10:	IF ip_state = BYTE#3 THEN (* Bei IP_Control anmelden *)
		url_length := LEN(domain_copy);
		char_count := 17 + url_length; (* sendebuffer initialisieren *)
		FOR i := 0 TO char_count DO
			S_BUF.BUFFER[i] := BYTE#00;
		END_FOR;
		tid := UINT_TO_BYTE(BYTE_TO_UINT(tid) + UINT#1);
		S_BUF.BUFFER[01] := tid; (* Transaction ID lowbyte *)
		S_BUF.BUFFER[02] := BYTE#16#01; (* Flags: highbyte *)
		S_BUF.BUFFER[05] := BYTE#16#01; (* Questions: lowbyte *)
		i := url_length + 12;	(* den servernamen von hinten nach vorne bearbeiten *)
		char_count := 0;
		WHILE i > 12 DO
			char := CODE(STR:=domain_copy,POS:=i - 12);
			IF char = BYTE#46 THEN (* prüfe auf haupt/sub domänen namens-teiler "." *)
				S_BUF.BUFFER[i] := INT_TO_BYTE(char_count); (* anstelle des teilers "." wird die länge des erkannten haupt/sub domänennames eingetragen *)
				char_count := 0;
			ELSE
				S_BUF.BUFFER[i] := char; (* char in buffer eintragen *)
				char_count := char_count + 1; (* anzahl char zählen *)
			END_IF;
			i := i - 1;
		END_WHILE;
		S_BUF.BUFFER[i] := INT_TO_BYTE(char_count); (* längenangabe des ganz linken (ersten) domänennamens eintragen *)
		i := url_length + 15; (* position hinter dem servernamen *)
		S_BUF.BUFFER[i] := BYTE#01; (* Type: A Hostaddress lowbyte *)
		i := i + 2;
		S_BUF.BUFFER[i] := BYTE#01; (* Class: IN lowbyte *)
		i := i + 1;
		(* IP Datenverkehr einrichten *)
		IP_C.C_PORT := WORD#53; (* Portnummer eintragen *)
		IP_C.C_IP := IP4_DNS; (* IP eintragen *)
		IP_C.C_MODE := BYTE#1; (* Mode: UDP+AKTIV+PORT+IP *)
		IP_C.C_ENABLE := TRUE; (* Verbindungsaufbau freigeben *)
		IP_C.TIME_RESET := TRUE; (* Zeitueberwachung rücksetzen *)
		IP_C.R_OBSERVE  := TRUE; (* Datenempfang ueberwachen *)
		S_BUF.SIZE := INT_TO_UINT(i); (* sendelänge eintragen *)
		R_BUF.SIZE := UINT#0; (* Empfangslänge rücksetzen *)
		state := 30;

        		(*####################  DEBUG-MESSAGE  ###################################*)
        		(*IF _debug_enable THEN
            		LOG_CL.NEW_MSG := 'DNS: S10 SEND';
            		LOG_MSG();
        		END_IF;*)
        		(*########################################################################*)
	END_IF;

30:	IF IP_C.ERROR <> DWORD#00 THEN
		ERROR := IP_C.ERROR;
		state := 99;
        		(*####################  DEBUG-MESSAGE  ###################################*)
        		(*IF _debug_enable THEN
            		LOG_CL.NEW_MSG := 'DNS: S30 ERROR ~1';
            		LOG_CL.PRINTF[1]  := DWORD_TO_STRING(ERROR);
            		LOG_MSG();
        		END_IF;*)
        		(*########################################################################*)

	ELSIF (S_BUF.SIZE = UINT#0) AND (tid = R_BUF.BUFFER[1]) AND (R_BUF.SIZE >= INT_TO_UINT(34 + url_length)) THEN	(* prüfe ob antwort telegramm die richtige Transaction-ID und mindestlänge hat *)
		ERROR := BYTE_TO_DWORD(R_BUF.BUFFER[3] AND BYTE#2#0000_1111); (* prüfe Return code der Flags. 4 bits *)
		IF ERROR = DWORD#00 THEN
			anc := R_BUF.BUFFER[7]; (* Anzahl der Answer-RR *)
			IP_C.R_OBSERVE := FALSE; (* Datenempfang ueberwachen *)
			state := 40;
		ELSE
			state := 99;
		END_IF;
	END_IF;

40:	IF anc > 0 THEN
		anc := anc - 1;
		WHILE i < R_BUF.SIZE DO
			x := R_BUF.BUFFER[i];
			IF rr_stop = FALSE THEN
				IF x > BYTE#63 THEN (* zeiger auf namen *)
					i := i + 1;
					rr_stop := TRUE;
				ELSIF x= BYTE#0 THEN (* namens ende *)
					rr_stop := TRUE;
				ELSE
					i := i + x; (* namen *)
				END_IF;
				i := i + 1;
			ELSE
				rr_stop := FALSE;
				IF R_BUF.BUFFER[i+1] = BYTE#1 AND R_BUF.BUFFER[i+3] = BYTE#1 THEN (* Type A / Class IN *)
					i := i + 4;
					ttl_tmp := DWORD_OF_BYTE(R_BUF.BUFFER[i],R_BUF.BUFFER[i+1],R_BUF.BUFFER[i+2],R_BUF.BUFFER[i+3]); (* Time to live *)
					i := i + 6;
					IF ttl_tmp >= ttl_last THEN (* TTL ist länger *)
						ttl_last := ttl_tmp;
						IP4 := DWORD_OF_BYTE(R_BUF.BUFFER[i],R_BUF.BUFFER[i+1],R_BUF.BUFFER[i+2],R_BUF.BUFFER[i+3]); (* IP-Adresse *)
					END_IF;
					i := i + 4;
				ELSE
					i := i + 9;
					i := i + R_BUF.BUFFER[i] + 1; (* offset zu nächsten Block *)
				END_IF;
				EXIT;
			END_IF;
		END_WHILE;
	ELSE
		IF IP4 > DWORD#0 THEN (* gültige RR mit IP gefunden *)
			DONE := TRUE;
            		(*####################  DEBUG-MESSAGE  ###################################*)
            		(*IF _debug_enable THEN
                			LOG_CL.NEW_MSG := 'DNS: S40 OK';
                			LOG_MSG();
            		END_IF;*)
            		(*########################################################################*)
		ELSE
			ERROR := DWORD#255; (* Daten fehlerhaft - keine IP-Adresse vorhanden *)
		END_IF;
		state := 99;
	END_IF;

99:	R_BUF.SIZE := UINT#0; (* Empfangslänge rücksetzen *)
	ip_state := BYTE#4; (* Abmelden *)
	state := 00;

END_CASE;

activate_last := ACTIVATE; (* letzten Status sichern zur Flankenerkennung *)
IP_FIFO(FIFO:=IP_C.FIFO,STATE:=ip_state,ID:=ip_id); (* IP_FIFO *)

(* revision history

ks	18. oct. 2008	rev 1.0
	original version

ks	20. oct. 2009	rev 1.1
	unbenutzten code entfernt, all buffer base 0

ks	20. dec. 2010	rev 1.2
	parsing nach rfc1305

ks	26. jul. 2011	rev 1.3
	verbesserte ip-auswertung , neue fehlermeldung
*)


(*----------------------------------------------------------------------------------------------------------------*)
(* Flags: 0x0100 (Standard query)                                                                                            *)
(* 0... .... .... .... = Response: Message is a query                                                                   *)
(* .000 0... ....  = Opcode: Standard query (0)                                                                          *)
(* .... ..0. .... .... = Truncated: Message is not truncated                                                          *)
(* .... ...1 .... .... = Recursion desired: Do query recursively                                                    *)
(* .... .... .0.. .... = Z: reserved (0)                                                                                                  *)
(* .... .... ...0 .... = Non-authenticated data OK: Non-authenticated data is unacceptable *)
(*-----------------------------------------------------------------------------------------------------------------*)

(*      0  1  2  3  4  5  6  7  8  9  0  1  2  3  4  5  *)
(*    +--+--+--+--+--+--+--+--+--+--+--+--+--+--+--+--+ *)
(*    |                      ID                       | idx: 0/1   *)
(*    +--+--+--+--+--+--+--+--+--+--+--+--+--+--+--+--+ *)
(*    |QR|   Opcode  |AA|TC|RD|RA|   Z    |   RCODE   | idx: 2/3   *)
(*    +--+--+--+--+--+--+--+--+--+--+--+--+--+--+--+--+ *)
(*    |                    QDCOUNT                    | idx: 4/5   *)
(*    +--+--+--+--+--+--+--+--+--+--+--+--+--+--+--+--+ *)
(*    |                    ANCOUNT                    | idx: 6/7   *)
(*    +--+--+--+--+--+--+--+--+--+--+--+--+--+--+--+--+ *)
(*    |                    NSCOUNT                    | idx: 8/9   *)
(*    +--+--+--+--+--+--+--+--+--+--+--+--+--+--+--+--+ *)
(*    |                    ARCOUNT                    | idx: 10/11 *)
(*    +--+--+--+--+--+--+--+--+--+--+--+--+--+--+--+--+ *)

(*
Errorcodes  Description	References 
000	No error. 		 	The request completed successfully.
001	Format error. 		The name server was unable to interpret the query. 
002	Server failure.  	The name server was unable to process this query due to a problem with the name server. 
003	Name Error. 	 	Meaningful only for responses from an authoritative name server, this code signifies that the domain name referenced in the query does not exist.
004	Not Implemented. 	The name server does not support the requested kind of query.
005	Refused. 			The name server refuses to perform the specified operation for policy reasons.
  						 For example, a name server may not wish to provide the information to the particular requester, or a name server may not wish to perform a particular operation (e.g., zone transfer) for particular data.
006	YXDomain.			Name Exists when it should not. 
007	YXRRSet. RR			Set Exists when it should not. 
008	NXRRSet. RR			Set that should exist does not. 
009	NotAuth.			Server Not Authoritative for zone. 
010	NotZone,			Name not contained in zone. 
255	Timeout				No Response  
   

beispiel einer DNS Request von google.at
ein request mit 3 Answer-Blocks


Domain Name System (response)
[Request In: 3]
[Time: 0.027533000 seconds]
Transaction ID: 0x5e1a
Flags: 0x8180 (Standard query response, No error)
1... .... .... .... = Response: Message is a response
.000 0... .... .... = Opcode: Standard query (0)
.... .0.. .... .... = Authoritative: Server is not an authority for domain
.... ..0. .... .... = Truncated: Message is not truncated
.... ...1 .... .... = Recursion desired: Do query recursively
.... .... 1... .... = Recursion available: Server can do recursive queries
.... .... .0.. .... = Z: reserved (0)
.... .... ..0. .... = Answer authenticated: Answer/authority portion was not authenticated
.... .... .... 0000 = Reply code: No error (0)
Questions: 1
Answer RRs: 3
Authority RRs: 0
Additional RRs: 0

Queries
google.at: type A, class IN
Name: google.at
Type: A (Host address)
Class: IN (0x0001)

Answers
google.at: type A, class IN, addr 72.14.221.104
Name: google.at
Type: A (Host address)
Class: IN (0x0001)
Time to live: 19 minutes, 9 seconds
Data length: 4
Addr: 72.14.221.104

google.at: type A, class IN, addr 66.249.93.104
Name: google.at
Type: A (Host address)
Class: IN (0x0001)
Time to live: 19 minutes, 9 seconds
Data length: 4
Addr: 66.249.93.104

google.at: type A, class IN, addr 216.239.59.104
Name: google.at
Type: A (Host address)
Class: IN (0x0001)
Time to live: 19 minutes, 9 seconds
Data length: 4
Addr: 216.239.59.104
*)

END_FUNCTION_BLOCK

// ---- oscat_basic/POUs/String/CHR_TO_STRING.TcPOU
FUNCTION CHR_TO_STRING : STRING(1)
VAR_INPUT
	C : BYTE;
END_VAR
VAR
	PT : POINTER TO BYTE;
END_VAR

(*
version 1.3	17. dec. 2008
programmer 	hugo
tested by	oscat

CHR creates a character from a byte input and stuffs it in a one character length string.

*)

PT := ADR(CHR_TO_STRING);
PT^ := C;
pt := pt + 1;
pt^ := 0;

(* revision history
hm	16 jan 2007		rev 1.0
	original version

hm	4. feb. 2008	rev 1.1
	return string would not be terminated properly

hm	29. mar. 2008	rev 1.2
	changed STRING to STRING(1)

hm	17. dec. 2008	rev 1.3
	changed name of function from chr to chr_to_string
*)

END_FUNCTION

// ---- beckhoff_network/POUs/DEMO/FTP_CLIENT_DEMO.TcPOU
PROGRAM FTP_CLIENT_DEMO
VAR
	FTP_CLIENT: FTP_CLIENT;
	ftp_activate: BOOL;
	ftp_done: BOOL;
	ftp_busy: BOOL;
	ftp_error_c: DWORD;
	ftp_error_t: BYTE;
	ftp_url: STRING := 'ftp://581920:123456@oscat.atwebpages.com:2000/subordner/';
	ftp_filename: STRING := '0100kb.bin';
	ftp_download: BOOL := TRUE;
	ftp_activ: BOOL := FALSE;
	file_delete: BOOL := FALSE;
	ftp_timeout: TIME := T#30s;
	zeit : TIME := T#30s;
	stop: BOOL;
	start: BOOL :=TRUE ;
	reset: BOOL;
	error: DWORD;
	ok: DWORD;
	CLK_PRG_1: CLK_PRG;
	COUNT_DR_1: COUNT_DR;
	COUNT_DR_2: COUNT_DR;
END_VAR
VAR // added by the converter: edge detectors and wires of the graphical bodies
    _w1, _w2 : ANY;
END_VAR

ftp_client(
    ACTIVATE := ftp_activate,
    FILENAME := ftp_filename,
    FTP_URL := ftp_url,
    FTP_DOWNLOAD := ftp_download,
    FTP_ACTIV := ftp_activ,
    FILE_DELETE := file_delete,
    TIMEOUT := ftp_timeout,
    DNS_IP4 := _w1,
    PLC_IP4 := _w2);
ftp_done := ftp_client.DONE;
ftp_busy := ftp_client.BUSY;
ftp_error_c := ftp_client.ERROR_C;
ftp_error_t := ftp_client.ERROR_T;
CLK_PRG_1(_in1 := zeit); // CLK_PRG
ftp_activate := CLK_PRG_1._out1 AND NOT stop AND start OR reset;
stop := ftp_error_t <> 0;
COUNT_DR_1(_in3 := stop); // COUNT_DR
error := COUNT_DR_1._out1;
COUNT_DR_2(_in3 := ftp_done); // COUNT_DR
ok := COUNT_DR_2._out1;
_w1 := DWORD_OF_BYTE(8, 8, 8, 8);
_w2 := DWORD_OF_BYTE(10, 145, 72, 57);

END_PROGRAM

// ---- beckhoff_network/POUs/NETWORK/FTP_CLIENT.TcPOU
FUNCTION_BLOCK FTP_CLIENT
VAR_INPUT
	ACTIVATE : BOOL;
	FILENAME : STRING;
	FTP_URL : STRING(STRING_LENGTH);
	FTP_DOWNLOAD : BOOL;
	FTP_ACTIV : BOOL;
	FILE_DELETE : BOOL;
	TIMEOUT : TIME;
	DNS_IP4 : DWORD;
	PLC_IP4 : DWORD;
END_VAR
VAR_OUTPUT
	DONE : BOOL;
	BUSY : BOOL;
	ERROR_C : DWORD;
	ERROR_T : BYTE;
END_VAR
VAR
	IP_C1 : IP_C; (* IP_Control Verwaltungsstruktur *)
	IP_C2 : IP_C; (* IP_Control Verwaltungsstruktur *)
	S_BUF1 : NETWORK_BUFFER;
	S_BUF2 : NETWORK_BUFFER;
	R_BUF1 : NETWORK_BUFFER;
	R_BUF2 : NETWORK_BUFFER;
	URL_DATA : url;
	DNS_CLIENT : DNS_CLIENT;
	IPC1 : IP_CONTROL;
	IPC2 : IP_CONTROL;
	FS : FILE_SERVER;
	FSD : FILE_SERVER_DATA;

	activate_last : BOOL;
	step : INT;
	snd_step : INT;
	snd_text :	STRING(STRING_LENGTH);
	rcv_text :	STRING(STRING_LENGTH);
	rcv_state : INT;
	TON_WAIT : TON;
	last_step : INT;
	next_step : INT;
	idx1 : INT;
	idx2 : INT;
	str1 : STRING(STRING_LENGTH);
	str2 : STRING(STRING_LENGTH);
	ftp_path : STRING;
	byar : ARRAY [0..5] OF BYTE;
	dw_tmp : DWORD;
	w_tmp : WORD;
	fpd : FILE_PATH_DATA;
	timeout2 : TIME;
	timeout3 : TIME;
	ftp_file_size : UDINT;
	ip_c1_red_disable : BOOL; (* IP_CONTROL 1 - Remote Disconnect Error unterdrücken *)
	ip_c2_red_disable : BOOL; (* IP_CONTROL 1 - Remote Disconnect Error unterdrücken *)

	(*LOG_MSG : LOG_MSG;
	_debug_enable : BOOL := FALSE;*)

END_VAR
(*
version 1.2		11.may 2011
programmer		ks
tested by			ks

FTP_CLIENT dient zum senden und empfangen von dateien von einem FTP-Server.



110 Restart marker reply 										Markierung für Wiederaufnahme der Übertragung 
120 Service ready in x minutes 									Dienst steht in x Minuten zu Verfügung 
125 Data connection already open; 								transfer starting Datenverbindung besteht bereits; beginne mit der Übertragung 
150 File status okay; about to open data connection 					Dateistatus OK; Datenverbindung wird aufgebaut 
200 Command okay 											Befehl OK 
202 Command not implemented 									Befehl nicht implementiert 
211   														Antwort für Systemstatus oder Hilfefunktion des Systems 
212   														Verzeichnisstatus 
213   														Dateistatus 
214   														Meldung der Hilfefunktion 
215 NAME system type 										Angabe des Systemtyps 
220 Service ready for new user 									Dienst bereit für neuen Benutzer 
221 Service closing control connection 							Steuerverbindung des Dienstes wird getrennt; Benutzer wird abgemeldet 
225 Data connection open; no transfer in progress 					Datenverbindung hergestellt; derzeit keine Übertragung 
226 Closing data connection. Requested file action successful 		Datenverbindung wird getrennt 
227 Entering Passive Mode 										Passiver Modus aktiviert 
230 User logged in, proceed 									Benutzer angemeldet, bitte fortfahren 
250 Requested file action okay, completed 						Angeforderter Vorgang OK, beendet 
257 "PATH" created 											"PFAD" wurde erstellt 
331 User name okay, need password 							Benutzername OK, Kennwort erforderlich 
332 Need account for login 										Benutzerkonto zur Anmeldung erforderlich 
350 Requested file action pending further information 				Mehr Informationen für Dateivorgang erforderlich 
421 Service not available, closing control connection 				Dienst nicht verfügbar, Steuerverbindung wird getrennt 
425 Can't open data connection 									Datenverbindung kann nicht hergestellt werden 
426 Connection closed; transfer aborted Verbindung getrennt; 		Übertragung abgebrochen 
450 Requested file action not taken; File unavailable 				Angeforderter Dateivorgang wurde nicht ausgeführt; Datei nicht verfügbar 
451 Requested action aborted: local error in processing 				Angeforderter Vorgang abgebrochen: Lokaler Fehler bei der Bearbeitung 
452 Requested action not taken; Insufficient storage space in system 	Angeforderter Vorgang nicht ausgeführt; Nicht genügend Speicherplatz auf System 
500 Syntax error 												Befehl nicht erkannt 
501 Syntax error in parameters or arguments 						Syntaxfehler bei den Parametern 
502 Command not implemented 									Befehl nicht implementiert 
503 Bad sequence of commands 								Ungültige Befehlsabfolge 
504 Command not implemented for that parameter 					Befehl für diesen Parameter nicht implementiert 
530 Not logged in 												Nicht angemeldet 
532 Need account for storing files 								Zum Speichern von Dateien Anmeldung erforderlich 
550 Requested file action not taken; File unavailable Angeforderter 	Dateivorgang wurde nicht ausgeführt; Datei nicht verfügbar 
551 Requested action aborted: page type unknown 					Angeforderter Vorgang abgebrochen: Unbekannter Seitentyp 
552 Requested file action aborted: Exceeded storage allocation 		Angeforderter Dateivorgang abgebrochen: Nicht genügend Platz in aktuellem Verzeichnis oder Datensatz 
553 Requested action not taken: File name not allowed 				Angeforderter Vorgang nicht ausgeführt: Unzulässiger Dateiname 

#########################
ERROR_T

1 = DNS_CLIENT
2 = FTP Steuerkanal
3 = FTP Datenkanal
4 = FILE_SERVER
5 = Ablaufstörung
#########################

*)

CASE step OF

00:	IF ACTIVATE AND NOT activate_last THEN
		ftp_file_size := UDINT#0;
		TIMEOUT := MAX(T#10s,TIMEOUT);
		timeout2 := TIMEOUT + T#1s;
		timeout3 := TIMEOUT / 2;
		DONE := FALSE;
		ip_c1_red_disable := FALSE;
		ip_c2_red_disable := FALSE;
		ERROR_C := DWORD#0;
		ERROR_T := BYTE#0;
		FSD.ERROR := BYTE#0;
		URL_DATA := STRING_TO_URL(STR:=FTP_URL,DEFAULT_PROTOCOL:='',DEFAULT_PATH:='/');
		IF LEN(URL_DATA.USER) = 0 THEN
			URL_DATA.USER := 'Anonymous';
			URL_DATA.PASSWORD := 'User@';
		END_IF;

		FILE_PATH_SPLIT(FILENAME:=FILENAME,X:=fpd); (* Datei-Path zerlegen *)
		str1 := fpd.FILENAME; (* zwischenspeichern *)
		FILE_PATH_SPLIT(FILENAME:=URL_DATA.PATH,X:=fpd); (* FTP-Path zerlegen *)
		IF LEN(fpd.FILENAME) = 0 THEN (* wenn FTP-Path keinen Dateinamen enthält , dann den Namen der lokalen Datei benutzen *)
			ftp_path := CONCAT(URL_DATA.PATH,str1);
		ELSE
			ftp_path := URL_DATA.PATH;
		END_IF;
		step := 10;
	END_IF;

10:	IF DNS_CLIENT.DONE THEN
		step := 20;
	ELSIF DNS_CLIENT.ERROR <> DWORD#0 THEN
		ERROR_C := DNS_CLIENT.ERROR;
		ERROR_T := BYTE#1;
		step := 980;
	END_IF;

20:	(* FTP Steuerkanal einrichten *)
	IP_C1.C_PORT := WORD#21; (* Portnummer eintragen *)
  	IP_C1.C_IP := DNS_CLIENT.IP4; (* IP eintragen *)
  	IP_C1.C_MODE := BYTE#0; (* Mode: TCP+ACTIV+PORT *)
  	IP_C1.TIME_RESET := TRUE; (* Zeitueberwachung rücksetzen *)
  	IP_C1.C_ENABLE := TRUE; (* Verbindungsaufbau freigeben *)
  	IP_C1.R_OBSERVE := TRUE; (* Empfangsueberwachung *)
	R_BUF1.SIZE := UINT#0;

  	IP_C2.C_ENABLE   := FALSE; (* Verbindungsaufbau sperren *)
	step := 30;

30:	IF rcv_state = 220 THEN (* 220 = Service ready for new user *)
		snd_text := CONCAT('USER ',URL_DATA.USER);
		next_step := 40;
	END_IF;

40:	IF rcv_state = 331 THEN (* 331 = User name okay, need password *)
		snd_text := CONCAT('PASS ',URL_DATA.PASSWORD);
		next_step := 50;
	ELSIF rcv_state = 230 THEN (* 230 = User logged in, proceed *)
		next_step := 50;
	ELSIF rcv_state = 220 THEN (* 220 = Service ready for new user *)
		next_step := 20; (* WORK verbindung sollte ab/aufgebaut werden *)
	END_IF;

50:	IF rcv_state = 230 THEN (* 230 = User logged in, proceed *)
		snd_text := 'TYPE I';  (* binären Modus aktivieren *)
		next_step := 54;
	END_IF;

54:	IF rcv_state = 200 THEN (* 200 = Command okay *)
		IF FTP_DOWNLOAD THEN (* Datei von FTP Empfangen *)
			snd_text := CONCAT('SIZE ', ftp_path); (* SIZE /PFAD/FILENAME *)
			next_step := 56;
		ELSE
			step := 60;
		END_IF;
	END_IF;

56:	IF rcv_state = 213 THEN (* 213 Filesize *)
		str1 := ELEMENT_GET(SEP:=BYTE#32,POS:=1,ELEMENT:=rcv_text);
		ftp_file_size := STRING_TO_UDINT(str1); (* Dateigroesse in bytes gestimmen *)
		step := 60;
	END_IF;

60:	IF FTP_ACTIV THEN (* FTP Server aktiv *)
		IF URL_DATA.PORT = WORD#0 THEN
			URL_DATA.PORT := WORD#20; (* Standard Datenkanal *)
		END_IF;
		str2 := '';
		dw_tmp := PLC_IP4;
		FOR idx1 := 0 TO 5 DO
			IF idx1 = 4 THEN
				dw_tmp := ROR(WORD_TO_DWORD(URL_DATA.PORT),8);
			ELSE
				dw_tmp := ROL(dw_tmp,8);
			END_IF;
			str2 := CONCAT(str2,BYTE_TO_STRING(DWORD_TO_BYTE(dw_tmp)));
			IF idx1 < 5 THEN
				str2 := CONCAT(str2,',');
			END_IF;
		END_FOR;
		dw_tmp := DNS_CLIENT.IP4; (* IP eintragen *)
		w_tmp := URL_DATA.PORT; (* Port Nummer des Datenkanals *)
		snd_text := CONCAT('PORT ',str2); (* FTP Server in den aktiv-mode schalten *)
		next_step := 80;
	ELSE
		snd_text := 'PASV';  (* FTP Server in den passiv-mode schalten *)
		next_step := 70;
	END_IF;
	step := 999; (* Warten auf next_step *)

70:	IF rcv_state = 227 THEN (* 227 = Entered Passive Mode (213,202,225,43,212,186) *)
		idx1 := FIND(rcv_text , '(' );
		idx2 := FIND(rcv_text , ')' );
		IF idx1 > 0 AND idx2 > idx1+1 THEN
			str1 := MID(rcv_text, idx2 - idx1 - 1, idx1+1);
			FOR idx1 := 0 TO 5 DO
				str2 := ELEMENT_GET(SEP:=BYTE#44,POS:=idx1,ELEMENT:=str1);
				byar[idx1] := STRING_TO_BYTE(str2);
			END_FOR;
			dw_tmp := DWORD_OF_BYTE(byar[0],byar[1],byar[2],byar[3]); (* IP Adresse des Datenkanals *)
			w_tmp := WORD_OF_BYTE(byar[4],byar[5]); (* Port Nummer des Datenkanals *)
		END_IF;
		step := 100;
	END_IF;

80:	IF rcv_state = 200 THEN (* 200 = PORT command successful *)
		step := 100;
	END_IF;

100:IP_C2.C_MODE := SEL(FTP_ACTIV,BYTE#0,BYTE#2); (* Aktiv = Mode 2: TCP+PASSIV+PORT / passiv = Mode 0: TCP+ACTIV+PORT *)
	IP_C2.C_IP := dw_tmp; (* IP Adresse des Datenkanals *)
	IP_C2.C_PORT := w_tmp; (* Port Nummer des Datenkanals *)
  	IP_C2.TIME_RESET := TRUE; (* Zeitueberwachung rücksetzen *)
  	IP_C2.C_ENABLE := TRUE; (* Verbindungsaufbau freigeben *)
	IP_C2.R_OBSERVE := FALSE; (* Empfangsueberwachung *)
	R_BUF2.SIZE := UINT#0;
	step := 120;

120:IF IP_C2.C_STATE > BYTE#127 THEN (* FTP Datenkanal aufgebaut *)
		IF FTP_DOWNLOAD THEN (* File von FTP empfangen *)
			IP_C2.MAILBOX[3] := BYTE#1; (* IP Empfang sperren *)
			step := 400;
		ELSE
			snd_text := 'STOR ';
			next_step := 140;
			snd_text := CONCAT(snd_text, ftp_path); (* STORE /PFAD/FILENAME *)
			step := 999; (* Warten auf next_step *)
		END_IF;
	END_IF;

(* ============== File an FTP senden ================ *)

140:IF rcv_state = 125 OR rcv_state = 150 THEN (* 125 = Data connection already open / 150 = File status okay; about to open data connection *)
		step := 160;
	END_IF;

160:FSD.FILENAME := FILENAME; (* Dateiname *)
	FSD.MODE := BYTE#1; (* vorhandene Datei zum lesen öffnen *)
	FSD.OFFSET := UDINT#0; (* Start bei Dateianfang *)
	FSD.AUTO_CLOSE := T#0s; (* kein Auto-Close verwenden *)
	S_BUF2.SIZE := UINT#65535; (* maximale länge einlesen *)
	IP_C2.MAILBOX[2] := BYTE#1; (* IP Senden blockieren *)
	step := 200;

200:IF FSD.MODE = BYTE#0 AND FSD.ERROR = BYTE#0 THEN
		IP_C2.MAILBOX[2] := BYTE#0; (* IP Senden erlauben *)
		step := 210;
	END_IF;

210:IF S_BUF2.SIZE = UINT#0 THEN (* warten bis alle daten gesendet sind *)
		IF FSD.FILE_SIZE - FSD.OFFSET > UDINT#0 THEN
			FSD.MODE := BYTE#1; (* vorhandene Datei zum lesen öffnen *)
			S_BUF2.SIZE := UINT#65535; (* maximale länge einlesen *)
			IP_C2.MAILBOX[2] := BYTE#1; (* IP Senden blockieren *)
			step := 200;
		ELSE
			IP_C2.C_ENABLE := FALSE; (* FTP Datenkanal schliessen *)
			step := 300;
		END_IF;
	END_IF;

300:IF rcv_state = 226 THEN (* 226 Closing data connection. Requested file action successful  *)
		snd_text := 'QUIT';
		ip_c1_red_disable := TRUE;
		next_step := 320;
	END_IF;

320:IF rcv_state = 221 OR TON_WAIT.ET > timeout3  THEN (* 221 Service closing control connection *)
		IP_C1.C_ENABLE := FALSE; (* FTP Steuerkanal schliessen *)
		IF FILE_DELETE THEN (* Datei nach transfer löschen *)
			FSD.MODE := BYTE#4; (* File Remove *)
			step := 340;
		ELSE
			step := 900;
		END_IF;
	END_IF;

340:IF FSD.MODE = BYTE#0 AND FSD.ERROR = BYTE#0 THEN
		step := 900;
	END_IF;

(*  ============== File vom FTP Empfangen  ============== *)

400:snd_text := 'RETR ';
	next_step := 410;
	snd_text := CONCAT(snd_text, ftp_path); (* RETR /PFAD/FILENAME *)
	step := 999; (* Warten auf next_step *)

410:IF rcv_state = 125 OR rcv_state = 150 THEN (* 125 = Data connection already open / 150 = File status okay; about to open data connection *)
		IP_C2.R_OBSERVE := TRUE; (* Empfangsueberwachung *)
		step := 420;
	END_IF;

420:FSD.FILENAME := FILENAME; (* Dateiname *)
	FSD.MODE := BYTE#3; (* Datei neu anlegen *)
	FSD.OFFSET := UDINT#0; (* Start bei Dateianfang *)
	FSD.AUTO_CLOSE := T#0s; (* kein Auto-Close verwenden *)
	step := 460;

440:IF R_BUF2.SIZE > UINT#0 THEN (* warten bis daten empfangen wurden *)
		IP_C2.MAILBOX[3] := BYTE#1; (* IP Empfang blockieren bis Daten in Datei geschrieben wurden *)
		FSD.MODE := BYTE#3; (* Daten in Datei schreiben *)
		step := 460;
	ELSIF FSD.FILE_SIZE = ftp_file_size THEN (* Verbindung abgebaut ? , oder 226 = Closing data connection. Requested file action successful *)
		IP_C2.C_ENABLE := FALSE; (* FTP Datenkanal schliessen *)
		ip_c2_red_disable := TRUE;
		step := 700;
	END_IF;

460:IF FSD.MODE = BYTE#0 AND FSD.ERROR = BYTE#0 THEN (* warten bis Daten geschreiben wurden *)
		R_BUF2.SIZE := UINT#0; (* Daten löschen *)
		IP_C2.MAILBOX[3] := BYTE#0; (* IP Empfang wieder erlauben *)
		step := 440;
	END_IF;

(* ================================================== *)

700:IF rcv_state = 226 OR  TON_WAIT.ET > timeout3 THEN (* 226 Closing control connection. Requested file action successful  *)
		IF FTP_DOWNLOAD AND FILE_DELETE THEN (* FTP Download und File löschen ? *)
			snd_text := CONCAT('DELE ', ftp_path); (* DELE /PFAD/FILENAME *)
			next_step := 720;
		ELSE
			step := 740;
		END_IF;
	END_IF;

720:IF rcv_state = 250 THEN (* 250 Requested file action okay, completed *)
		step := 740;
	END_IF;

740:snd_text := 'QUIT';
	ip_c1_red_disable := TRUE;
	next_step := 760;
	step := 999; (* Warten auf next_step *)

760:IF rcv_state = 221 OR TON_WAIT.ET > timeout3 THEN (* 221 Service closing control connection  *)
		IP_C1.C_ENABLE := FALSE; (* FTP Steuerkanal schliessen *)
		IF NOT FTP_DOWNLOAD AND FILE_DELETE THEN (* FTP Upload und Datei nach transfer löschen *)
			FSD.MODE := BYTE#4; (* File Remove *)
			step := 780;
		ELSE
			step := 900;
		END_IF;
	END_IF;

780:IF FSD.MODE = BYTE#0 AND FSD.ERROR = BYTE#0 THEN
		step := 900;
	END_IF;

(* ================================================== *)

900:DONE := TRUE;
	step := 980;

980:IP_C1.C_ENABLE := FALSE; (* FTP Steuerkanal schliessen *)
	IP_C2.C_ENABLE := FALSE; (* FTP Datenkanal schliessen *)
	IP_C2.MAILBOX[2] := BYTE#0; (* IP Senden wieder erlauben *)
	IP_C2.MAILBOX[3] := BYTE#0; (* IP Empfang wieder erlauben *)
	S_BUF1.SIZE := UINT#0;
	S_BUF2.SIZE := UINT#0;
	R_BUF1.SIZE := UINT#0;
	R_BUF2.SIZE := UINT#0;
	ftp_file_size := UDINT#0;
	snd_step := 0;
	next_step := 0;
	FSD.MODE := BYTE#5; (* Datei schliessen *)
	step := 990;

990:IF IP_C1.C_STATE = BYTE#0 AND IP_C2.C_STATE = BYTE#0 AND FSD.FILE_OPEN = FALSE THEN
		step := 0;
	END_IF;

999: ; (* Dummy Schritt, warten bis neuer schritt durch "next_step" aktiv wird *)

END_CASE;

(* ++++++++++++++++++++++++++++++++++++++++++++++++++++++++++ *)

IF step >= 30 THEN
	IF R_BUF1.SIZE > UINT#0 THEN (* Daten wurden empfangen ? *)
		idx1 := UINT_TO_INT(R_BUF1.SIZE);
		REPEAT (* zeilenterminierung erkennen und echtes TEXT-Ende bestimmen *)
			idx1 := idx1 - 1;
		UNTIL idx1 = 0 OR R_BUF1.BUFFER[idx1] >= BYTE#32 (* TRUE = EXIT *)
		END_REPEAT;
		idx1 := idx1 + 1; (* index auf SIZE umrechnen *)
		rcv_text := BUFFER_TO_STRING(PT:=ADR(R_BUF1.BUFFER),SIZE:=idx1,START:=0,STOP:=STRING_LENGTH-1);
		IF LEN(rcv_text) >= 3 THEN (* Statuscode prüfen und auswerten *)
			str1 := LEFT(rcv_text,3);
			IF IS_NUM(STR:=str1) THEN (* enthält nur Zahlen ? *)
				rcv_state := STRING_TO_INT(str1);
			END_IF;
			IP_C1.R_OBSERVE := FALSE;
		END_IF;
		R_BUF1.SIZE := UINT#0; (* daten löschen *)

	        (*####################  DEBUG-MESSAGE  ###################################*)
	        (*IF _debug_enable THEN
	          LOG_CL.NEW_MSG := 'RCV: >~1<';
	          LOG_CL.PRINTF[1] := rcv_text;
	          LOG_MSG();
	        END_IF;*)
	        (*########################################################################*)

	END_IF;
END_IF;

(* automatisches Datensenden *)

CASE snd_step OF

00:	IF LEN(snd_text) > 0 THEN
	        (*####################  DEBUG-MESSAGE  ###################################*)
	        (*IF _debug_enable THEN
	          LOG_CL.NEW_MSG := 'SND: >~1<';
	          LOG_CL.PRINTF[1] := snd_text;
	          LOG_MSG();
	        END_IF;*)
	        (*########################################################################*)
		_STRING_TO_BUFFER(str:=snd_text,pos:=0,pt:=ADR(S_BUF1.BUFFER),size:=SIZEOF(S_BUF1.BUFFER)); (* String in puffer kopieren *)
		idx1 := LEN(snd_text);
		S_BUF1.BUFFER[idx1] := BYTE#16#0D;
		idx1 := idx1 + 1;
		S_BUF1.BUFFER[idx1] := BYTE#16#0A;
		idx1 := idx1 + 1;
		S_BUF1.SIZE := INT_TO_UINT(idx1); (* Sendelänge eintragen *)
		R_BUF1.SIZE := UINT#0; (* Empfangsbuffer rücksetzen *)
		IP_C1.R_OBSERVE := TRUE;
		rcv_state := 9999; (* letzen FTP Status löschen *)
		snd_text := '';
		snd_step := 10;
	END_IF;

10:	IF S_BUF1.SIZE = UINT#0 THEN (* warten bis alle daten gesendet sind *)
		step := next_step;
		snd_step := 0;
	END_IF;

END_CASE;

(* Globale Fehlerbehandlung für Haupt-Routine *)
IF ERROR_T = BYTE#0 AND step > 20 THEN (* noch kein Fehler gespeichert und Hauptroutine aktiv *)

	IF IP_C1.ERROR > DWORD#0 AND IP_C1.C_ENABLE AND NOT IP_C1.TIME_RESET THEN  (* IP Control 1 *)
		IF ip_c1_red_disable = FALSE OR IP_C1.ERROR <> DWORD#16#FD000000 THEN
			ERROR_C := IP_C1.ERROR;
			ERROR_T := BYTE#2;
			step := 980;
		END_IF;
	END_IF;

	IF IP_C2.ERROR > DWORD#0 AND IP_C2.C_ENABLE AND NOT IP_C2.TIME_RESET THEN  (* IP Control 2 *)
		IF ip_c2_red_disable = FALSE OR IP_C2.ERROR <> DWORD#16#FD000000 THEN
			ERROR_C := IP_C2.ERROR;
			ERROR_T := BYTE#3;
			step := 980;
		END_IF;
	END_IF;

	IF FSD.MODE = BYTE#0 THEN
		IF FSD.ERROR > BYTE#0 THEN
			ERROR_C := BYTE_TO_DWORD(FSD.ERROR);
			ERROR_T := BYTE#4; (* Dateizugriff *)
			step := 980;
		END_IF;
	END_IF;
END_IF;

IF TON_WAIT.Q THEN (* Ablaufstörung - Schrittkette *)
	ERROR_C := SHL(INT_TO_DWORD(step),16) OR INT_TO_DWORD(rcv_state); (* aktuellen Schritt und letzten FTP Status eintragen *)
	ERROR_T := BYTE#5;
	step := 980;
END_IF;

(* ######################################################## *)

DNS_CLIENT(IP_C:=IP_C1, S_BUF:=S_BUF1, R_BUF:=R_BUF1, DOMAIN:=URL_DATA.DOMAIN, IP4_DNS:= DNS_IP4, ACTIVATE:=step=10); (* DNS-Client *)
IPC1(IP:= DWORD#0, PORT:= WORD#0 , TIME_OUT:= TIMEOUT, IP_C:= IP_C1, S_BUF:= S_BUF1, R_BUF:= R_BUF1); (* FTP Steuerkanal *)
IPC2(IP:= DWORD#0, PORT:= WORD#0 , TIME_OUT:= TIMEOUT, IP_C:= IP_C2, S_BUF:= S_BUF2, R_BUF:= R_BUF2); (* FTP Datenkanal *)

TON_WAIT(IN:=step = last_step AND step > 0,PT:=timeout2);
last_step := step;
activate_last := ACTIVATE;
BUSY := step <> 0;

IF FTP_DOWNLOAD THEN (* FILE_SERVER *)
	FS(FSD:=FSD,PT:=R_BUF2); (* Datei von FTP empfangen *)
ELSE
	FS(FSD:=FSD,PT:=S_BUF2); (* Datei an FTP senden *)
END_IF;

(* revision history
ks	11. may 2011	rev 1.2
	ip_control - remote disconnect error ausblenden, und sonderbehandlung für pcworx

ks	06. apr. 2011	rev 1.1
	list_len und list_get durch element_count und element_get ersetzt

ks	01. jan. 2011	rev 1.0
	original version
*)

END_FUNCTION_BLOCK

// ---- oscat_basic/POUs/Logic/gate logic/WORD_OF_BYTE.TcPOU
FUNCTION WORD_OF_BYTE : WORD
VAR_INPUT
	B1 : BYTE;
	B0 : BYTE;
END_VAR


(*
version 1.4	18. jul. 2009
programmer 	hugo
tested by		tobias

this function creates a word from 2 individual bytes

*)

WORD_OF_BYTE := SHL(BYTE_TO_WORD(B1),8) OR BYTE_TO_WORD(B0);

(* revision history
hm	24. jan 2007	rev 1.0
	original version

hm	2. jan 2008	rev 1.1
	improved performance

hm	19. feb 2008	rev 1.2
	replaced and with or for better compatibility

hm	23. apr. 2008	rev 1.3
	reverse order of inputs to be more logical

hm	18. jul. 2009	rev 1.4
	added type conversions for compatibility reasons

*)

END_FUNCTION

// ---- beckhoff_network/POUs/DEMO/GET_WAN_IP_DEMO.TcPOU
PROGRAM GET_WAN_IP_DEMO
VAR
	GET_WAN_IP: GET_WAN_IP;
	IP_C: IP_C;
	S_BUF: NETWORK_BUFFER;
	R_BUF: NETWORK_BUFFER;
	IP_CONTROL_1: IP_CONTROL;
	activate: BOOL;
	done: BOOL;
	error_c: DWORD;
	error_t: BYTE;
	wan_ip: STRING;
	new_ip: BOOL;
END_VAR
VAR // added by the converter: edge detectors and wires of the graphical bodies
    _w1 : ANY;
END_VAR

GET_WAN_IP(ACTIVATE := activate, IP_C := IP_C, S_BUF := S_BUF, R_BUF := R_BUF);
done := GET_WAN_IP.DONE;
new_ip := GET_WAN_IP.NEW_IP4;
error_c := GET_WAN_IP.ERROR_C;
error_t := GET_WAN_IP.ERROR_T;
wan_IP := IP4_TO_STRING(IP4 := GET_WAN_IP.WAN_IP4);
// IP-Adresse des DNS-Server oder des DSL-Router
_w1 := DWORD_OF_BYTE(8, 8, 8, 8);
IP_CONTROL_1(IP := _w1, TIME_OUT := T#1s, IP_C := IP_C, S_BUF := S_BUF, R_BUF := R_BUF); // IP_CONTROL

END_PROGRAM

// ---- beckhoff_network/POUs/DEMO/INI_PARSER_BUF_DEMO.TcPOU
PROGRAM INI_PARSER_BUF_DEMO
VAR
	STATION_NAME : STRING;
	STATION_IP : STRING;
	SMTP_SERVER : STRING;
	SMTP_FROM :	STRING;

	IPB : INI_PARSER_BUF;
	FS : FILE_SERVER;
	FSD : FILE_SERVER_DATA;
	PT : NETWORK_BUFFER;
	section : INT;
	key : STRING(STRING_LENGTH);
	value : STRING(STRING_LENGTH);
	str : STRING(STRING_LENGTH);
	step : INT;
	result : BYTE;
	offset : UDINT;
	run : BYTE;
	done : BOOL;

	(*_debug_enable : BOOL := TRUE;
	LOG_MSG : LOG_MSG;*)
END_VAR

(* Demo-Programm: INI-Datei mittels Enumeration auswerten *)

(* ----- den nachfolgenden Textblock als datei "config.ini" auf der sps ablegen ---
# Demo - Initialisierungsdatei

[Station]
NAME=Test_Station_1
IP=192.168.178.1

[SMTP]
SERVER=test.server.de
FROM=test1@gmx.net
---------------------------------------------------------------------------------*)

CASE step OF

00:	IF NOT done THEN
	 	(* File_Daten einrichten  *)
		FSD.FILENAME := 'config.ini'; (* Dateiname *)
		FSD.MODE := 1; (* vorhandene Datei zum lesen öffnen *)
		FSD.OFFSET := 0; (* Start bei Dateianfang *)
		FSD.AUTO_CLOSE := T#0s; (* kein Auto-Close verwenden *)
		PT.SIZE := 65535; (* maximale länge einlesen *)
		step := 10;
	END_IF;

10:	IF FSD.MODE = 0 THEN (* Datei geöffnet ? *)
		OFFSET := 0; (* Start Offset vorgeben *)
		str := '';
		run := 3; (* key suchen *)
		step := 20;
	END_IF;

20:	IF run = 0 THEN
		(* ---------------------- Debug-Message ----------------------------*)
		(*IF _debug_enable THEN
			LOG_CL.NEW_MSG := 'IPBD: /key >~1< /value >~2< /offset ~3 /Run ~4 /Result ~5';
			LOG_CL.PRINTF[1] := key;
			LOG_CL.PRINTF[2] := value;
			LOG_CL.PRINTF[3] := UDINT_TO_STRING(OFFSET);
			LOG_CL.PRINTF[4] := BYTE_TO_STRING(run);
			LOG_CL.PRINTF[5] := BYTE_TO_STRING(result);
			LOG_MSG();
		END_IF;*)
		(* -----------------------------------------------------------------*)

		run := 3; (* vorbelegung -> naechsten key suchen *)

		IF result = 1 THEN (* neue Sektion gefunden *)
			IF key = 'Station' THEN
				section := 1;
			ELSIF key = 'SMTP' THEN
				section := 2;

			(* hier können weitere Section hinzugefügt werden *)

			ELSE
				section := 0; (* unbekannte sektion gefunden -> ignorieren *)
			END_IF;

		ELSIF result = 2 AND section > 0 THEN (* Key in einer bekannten sektion gefunden *)

			CASE section OF

			1:  (* Section: Station *)
				IF key = 'NAME' THEN
					STATION_NAME := value; (* Name *)
				ELSIF key = 'IP' THEN
					STATION_IP := value; (* IP-Adresse *)
				END_IF;

				(* hier können weitere Schlüsselsauswertungen hinzugefügt werden *)

			2:  (* Section: SMTP *)
				IF key = 'SERVER' THEN
					SMTP_SERVER := value; (* SMTP Server *)
				ELSIF key = 'FROM' THEN
					SMTP_FROM := value; (* SMTP Absender *)
				END_IF;

				(* hier können weitere Schlüsselsauswertungen hinzugefügt werden *)

			END_CASE;

		ELSIF result = 10 THEN (* nichts mehr gefunden *)
			run := 0; (* keine weitere INI Auswertung erwünscht *)
			FSD.MODE := 5; (* Datei schliessen *)
			step := 30;
		END_IF;
	END_IF;

30:	IF FSD.MODE = 0 THEN (* Datei geschlossen ? *)
		step := 0;
		done := TRUE;
	END_IF;

END_CASE;

IPB(STR:=str,RUN:=run,OFFSET:=OFFSET,KEY:=key,VALUE:=value,PT:=PT); (* INI PARAMETER BUF *)
result:=IPB.RESULT;

FS(FSD:=FSD,PT:=PT); (* FILE_SERVER *)

END_PROGRAM

// ---- beckhoff_network/POUs/DEMO/IP2GEO_DEMO.TcPOU
PROGRAM IP2GEO_DEMO
VAR
	IP_C: IP_C;
	S_BUF: NETWORK_BUFFER;
	R_BUF: NETWORK_BUFFER;
	IP_CONTROL_1: IP_CONTROL;
	CLK_PRG : CLK_PRG;
	IP2GEO_1: IP2GEO;
	GEO: IP2GEO_DATA;
	activate: BOOL := TRUE;
	done: BOOL;
	busy: BOOL;
	error_c: DWORD;
	error_t: BYTE;
END_VAR
VAR // added by the converter: edge detectors and wires of the graphical bodies
    _w1 : ANY;
END_VAR

CLK_PRG(_in1 := t#3h);
activate := CLK_PRG._out1;
IP2GEO_1(ACTIVATE := activate, IP_C := IP_C, S_BUF := S_BUF, R_BUF := R_BUF, GEO := GEO); // IP2GEO
busy := IP2GEO_1.BUSY;
done := IP2GEO_1.DONE;
error_c := IP2GEO_1.ERROR_C;
error_t := IP2GEO_1.ERROR_T;
// IP-Adresse des DNS-Server oder des DSL-Router
_w1 := DWORD_OF_BYTE(8, 8, 8, 8);
IP_CONTROL_1(IP := _w1, TIME_OUT := T#5s, IP_C := IP_C, S_BUF := S_BUF, R_BUF := R_BUF); // IP_CONTROL

END_PROGRAM

// ---- beckhoff_network/POUs/NETWORK/IP2GEO.TcPOU
FUNCTION_BLOCK IP2GEO
VAR_IN_OUT
	IP_C : IP_C; (* IP_Control Verwaltungsstruktur *)
	S_BUF : NETWORK_BUFFER;
	R_BUF : NETWORK_BUFFER;
	GEO : IP2GEO_DATA;
END_VAR
VAR_INPUT
	IP : DWORD;
	ACTIVATE : BOOL;
END_VAR
VAR_OUTPUT
	BUSY : BOOL;
	DONE : BOOL;
	ERROR_C : DWORD;
	ERROR_T : BYTE;
END_VAR
VAR
	CTRL : XML_CONTROL;
	XML_READER : XML_READER;
	URL_DATA : url;
	DNS_CLIENT : DNS_CLIENT;
	HTTP_GET : HTTP_GET;
	last_state : BOOL;
	value_int :	INT;
	value_real : REAL;
	v_real : REAL;
	state : INT;
END_VAR
(*

version 	1.1	07.oct. 2010
programmer 	ks
tested by	ks

IP2GEO ermittelt die aktuelle WAN-IP und die dazugehörigen geographischen Infos

zusatzinfos: http://www.worldtimezone.com/time/wtzresult.php?CiID=10182&forma=

example:

http://ipinfodb.com/ip_query.php?timezone=true&IP=

<?xml version="1.0" encoding="UTF-8" ?> 
- <Response>
  <Ip>85.127.218.109</Ip> 
  <Status>OK</Status> 
  <CountryCode>AT</CountryCode> 
  <CountryName>Austria</CountryName> 
  <RegionCode>09</RegionCode> 
  <RegionName>Wien</RegionName> 
  <City>Vienna</City> 
  <ZipPostalCode /> 
  <Latitude>48.2</Latitude> 
  <Longitude>16.3667</Longitude> 
  <TimezoneName>Europe/Vienna</TimezoneName> 
  <Gmtoffset>7200</Gmtoffset> 
  <Isdst>1</Isdst> 
  </Response>

*)

CASE state OF

00:
	IF ACTIVATE AND NOT last_state THEN
		state := 20;
		DONE := FALSE;
		BUSY := TRUE;
		ERROR_C := DWORD#0;
		ERROR_T := BYTE#0;
	END_IF;

20: (* URL for DNS UND HTTP-GET *)
	(* Example: http://ipinfodb.com/ip_query.php?ip=10.10.10.10 *)
	(* Example: http://ipinfodb.com/ip_query.php?timezone=true&IP=*)
	URL_DATA:=STRING_TO_URL(STR:='http://ipinfodb.com/ip_query.php?timezone=true&IP=',DEFAULT_PROTOCOL:='',DEFAULT_PATH:='');

	IF IP > DWORD#0 THEN
		URL_DATA.QUERY := CONCAT(URL_DATA.QUERY,IP4_TO_STRING(IP4:=IP));
	END_IF;

	state := 40;

40:
	IF DNS_CLIENT.DONE THEN
		state := 60;
	ELSIF (DNS_CLIENT.ERROR > DWORD#00) THEN
		(* Fehlerbehandlung *)
		ERROR_C := DNS_CLIENT.ERROR;
		ERROR_T := BYTE#01;
		state := 100;
	END_IF;

60:
	IF HTTP_GET.DONE THEN
		state := 80;
		CTRL.START_POS := HTTP_GET.BODY_START;
		CTRL.STOP_POS := HTTP_GET.BODY_STOP;
		CTRL.COMMAND := WORD#2#10000000_00011000; (* ONLY TEXT AND ATTRIBUTE *)
		CTRL.WATCHDOG := T#1ms;

	ELSIF (HTTP_GET.ERROR > DWORD#00) THEN
		(* Fehlerbehandlung *)
		ERROR_C := HTTP_GET.ERROR;
		ERROR_T := BYTE#02;
		state := 100;
	END_IF;

80:
	(* XML Daten seriell lesen *)
	XML_READER(CTRL:=CTRL,BUF:=R_BUF.BUFFER);
	IF CTRL.TYP < 98 THEN (* nur auswerten wenn kein Watchdog durchlauf *)
		(* automatische konvertierung in real und int ausführen *)
		value_int := 0;
		value_real := 0.0;
		IF LEN(CTRL.VALUE) <= 20 THEN
			v_real :=FLOAT_TO_REAL(FLT:=CTRL.VALUE);
			IF CHK_REAL(v_real) = 0 THEN (* !!! prüft auf gültigen REAL Wert, ansonsten stürzt Twincat ab !!!!  *)
				value_real := v_real;
				value_int := REAL_TO_INT(value_real);
			END_IF;
		END_IF;

		CASE UINT_TO_INT(CTRL.COUNT) OF

		07: GEO.IP4 := IP4_DECODE(STR:=CTRL.VALUE); (* IP-Adresse *)
		10: GEO.STATE := 'OK' = CTRL.VALUE; (* STATUS *)
		13: GEO.COUNTRY_CODE := CTRL.VALUE; (* Country-Code *)
		16: GEO.COUNTRY_NAME := CTRL.VALUE; (* Country-Name *)
		19: GEO.REGION_CODE := CTRL.VALUE; (* Region-Code *)
		22: GEO.REGION_NAME := CTRL.VALUE; (* Region-Name *)
		25: GEO.CITY := CTRL.VALUE; (* City *)
		31: GEO.GEO_LATITUDE := value_real; (* Latitude *)
		34: GEO.GEO_LONGITUDE := value_real; (* Longitude *)
		37: GEO.TIME_ZONE_NAME := CTRL.VALUE; (* TimeZone Name *)
		40: GEO.GMT_OFFSET := value_int; (* GMT OFFSET in Sekunden *)
		43: GEO.IS_DST := value_int > 0; (* Sommerzeit aktiv *)
		END_CASE;

	ELSIF CTRL.TYP = 99 THEN (* EXIT - letztes Element gelesen *)
		DONE := TRUE;
		state := 100;
	END_IF;

100:
	(* UNLOCK HTTP DATA *)
	IF (NOT HTTP_GET.DONE) THEN
		state := 0;
		BUSY := FALSE;
		DONE := ERROR_T = BYTE#0;
	END_IF;

END_CASE;

(* ---------------- DNS --------------- *)
DNS_CLIENT(	IP_C:=IP_C,
			S_BUF:=S_BUF,
			R_BUF:=R_BUF,
			DOMAIN:=URL_DATA.DOMAIN,
			IP4_DNS:=DWORD#00,
			ACTIVATE:=state=40 (* DNS Start *)
			);

(* nicht oder nicht direkt verwendete Parameter *)
(* 	DWORD :=DNS_CLIENT.IP4;
	BOOL  :=DNS_CLIENT.DONE;
	BYTE  :=DNS_CLIENT.ERROR; *)
(* -------------------------------------*)

(* ------------- HTTP_GET --------------- *)
HTTP_GET(	IP_C:=IP_C,
			S_BUF:=S_BUF,
			R_BUF:=R_BUF,
			IP4:=DNS_CLIENT.IP4,
			GET:=state=60,
			MODE:=BYTE#2, (* HTTP 1.1 mit persistenter Verbindung *)
			UNLOCK_BUF:=state=100,
			URL_DATA:=URL_DATA
			);

(* nicht oder nicht direkt verwendete Parameter *)
(*	STRING := HTTP_GET.HTTP_STATUS;
	UINT :=HTTP_GET.HEADER_START;
	UINT :=HTTP_GET.HEADER_STOP;
	UINT :=HTTP_GET.BODY_START;
	UINT :=HTTP_GET.BODY_STOP;
	BOOL :=HTTP_GET.DONE;
	BYTE :=HTTP_GET.ERROR;
*)
(* -------------------------------------*)

last_state := ACTIVATE;

(* revision history
ks	14. aug. 2009	rev 1.0
	original version

ks	07. oct. 2010	rev 1.1
	new url , ip2geo fields , REAL_CHECK
*)

END_FUNCTION_BLOCK

// ---- beckhoff_network/POUs/DEMO/MB_SERVER_DEMO.TcPOU
PROGRAM MB_SERVER_DEMO
VAR
	IP_CONTROL2_1: IP_CONTROL2;
	MB_SERVER_1: MB_SERVER;
	IP_C: IP_C;
	S_BUF: NETWORK_BUFFER_SHORT;
	R_BUF: NETWORK_BUFFER_SHORT;
	DATA: ARRAY [0..255] OF WORD;
	VMAP: ARRAY [1..10] OF VMAP_DATA;
END_VAR

MB_SERVER_1(
    DATA_SIZE := 10,
    ENABLE := TRUE,
    UDP := FALSE,
    IP_C := IP_C,
    S_BUF := S_BUF,
    R_BUF := R_BUF,
    VMAP := VMAP,
    DATA := DATA); // MB_SERVER
IP_CONTROL2_1(PORT := 502, TIME_OUT := T#2s, IP_C := IP_C, S_BUF := S_BUF, R_BUF := R_BUF); // IP_CONTROL2

END_PROGRAM

// ---- beckhoff_network/POUs/HARDWARE/IP_CONTROL2.TcPOU
FUNCTION_BLOCK IP_CONTROL2
VAR_IN_OUT
	IP_C : IP_C; (* IP_Control Verwaltungsstruktur *)
	S_BUF : NETWORK_BUFFER_SHORT; (* Externer Sendbuffer *)
	R_BUF : NETWORK_BUFFER_SHORT; (* Externer Receivebuffer *)
END_VAR
VAR_INPUT
	IP : DWORD; (* IP Adresse *)
	PORT : WORD; (* Port Nummer *)
	TIME_OUT : TIME; (* Ueberwachungszeit Connect / Send / Receive *)
END_VAR
VAR
	c_time : UDINT; (* CONNECT-Time (Zeit bei nicht vorhandener Verbindung) *)
	s_time : UDINT; (* SEND-Time    (Zeit seit letzten Datensenden) *)
	r_time : UDINT; (* RECEIVE-Time (Zeit seit letztem Datenempfang) *)

	c_enable : BOOL; (* Connect: freigabe *)
	c_ip : DWORD; (* Connect: aktuelle IP-Adresse *)
	c_ip_str : STRING(15);
	c_port : WORD; (* Connect: aktuelle Port-Nummer *)
	c_mode : BYTE; (* Connect: aktueller Mode UDP/TCP...... *)
	c_status : BYTE; (* Connect: Status (Errorcode) *)
	c_ready : BOOL; (* Connect: Verbindung aufgebaut *)
	c_ready_old : BOOL; (* Connect: letzter Zustand von c_ready für Flankenauswertung *)

	s_total : INT; (* Send: Gesamtanzahl Bytes zum senden *)
	s_cur_pos : INT; (* Send: aktuelle Sendeposition *)
	s_cur_size : INT; (* Send: aktuelle Sendegroesse *)
	s_max_size : INT; (* Send: maximale Telegrammlänge fuer Senden *)
	s_active : BOOL; (* Send: Daten senden ist aktiv *)
	s_status : BYTE; (* Send: Status (Errorcodes) *)
	s_ip_str : STRING(15);
	s_ip_exist : BOOL;

	r_status : BYTE; (* Receive: Status (Errorcodes) *)
	r_count : INT; (* Receive: Anzahl empfangener Bytes *)
	r_offset : INT; (* Receive: aktuelle Position in externen Receivebuffer *)
	r_max_size : INT; (* Receive: groesse des externen Empfangbuffers*)

	new_connection : BOOL; (* Neue Verbindungsparameter vorhanden *)
	tx : DWORD; (* letzter zeitwert *)
	error_time : DWORD; (* aktueller Timeout-Wert *)

	state: BYTE; (* schrittmerker für connect *)
	bytes_received : DINT;
	udp_mode : BOOL;

	socket : T_HSOCKET;
	server : T_HSOCKET;
	fbCreate	: FB_SocketUdpCreate;
	fbConnect : FB_SocketConnect;
	fbClose : FB_SocketClose;
	fbSendTo : FB_SocketUdpSendTo;
	fbReceiveFrom : FB_SocketUdpReceiveFrom;
	fbSend : FB_SocketSend;
	fbReceive : FB_SocketReceive;
	fbListen : FB_SocketListen;
	fbAccept : FB_SocketAccept;
	nErrId : UDINT;
	Send_Busy : BOOL;
	Send_Error : BOOL;
	Send_ErrId : UDINT;

	IPCR : IP_CONTROL_RESET;

	(*LOG_MSG : LOG_MSG;
	_debug_enable : BOOL := TRUE;
	debug_index : INT;
	debug_ID : INT;
	debug_lasterror : DWORD;
	state_last : INT;
	debug_last_id : INT := 255;*)
END_VAR

VAR CONSTANT
	STOP : BYTE := 0;
	UDP_INIT : BYTE:= 31;
	UDP_INIT_WAIT : BYTE:= 32;
	TC_INIT : BYTE := 51;
	TC_CONNECT : BYTE:= 52;
	TS_INIT : BYTE:= 53;
	TS_LISTEN_WAIT : BYTE:= 54;
	TS_ACCEPT : BYTE:= 55;
	TS_ACCEPT_WAIT : BYTE:= 56;
	C_CLOSE : BYTE := 190;
	C_CLOSE_WAIT : BYTE:= 191;
	C_CLOSE2 : BYTE := 192;
	C_CLOSE_WAIT2 : BYTE:= 193;
	C_WAIT : BYTE := 200;
	C_REC : BYTE := 210;
	C_REC_WAIT : BYTE := 211;
	C_SND : BYTE := 220;
	C_SND_WAIT1 : BYTE := 221;
	C_SND_WAIT2 : BYTE := 222;
END_VAR

(*

version 1.8		26. july. 2011
programmer 		ks
tested by			ks

IP_CONTROL ist ein Wrapper-Baustein um eine Hersteller neutrale Schnittstelle zum Ethernet zu schaffen


TYP 	TCP / UDP 	Aktiv / Passiv 		Port-Nummer erforderlich 	IP-Adresse erforderlich
0 		TCP 		Aktiv 			Ja 						Ja
1 		UDP 		Aktiv 			Ja 						Ja
2 		TCP 		Passiv 			Ja 						Ja (Adresse des aktiven Partners)
3 		UDP 		Passiv 			Ja 						Ja (Adresse des aktiven Partners)
4 		TCP 		Passiv 			Ja 						Nein (beliebiger aktiver Partner wird akzeptiert)
5 		UDP 		Passiv 			Ja 						Nein (beliebiger aktiver Partner wird akzeptiert)

*)

(* Bei PLC reset oder Programm Download werden alle alten Verbindungen geschlossen *)
IPCR();
IF NOT IPCR.READY THEN RETURN; END_IF;

(* ---------------------- Debug-Message ----------------------------*)
(*IF _debug_enable THEN
	IF IP_C.FIFO.ID > BYTE#0 THEN (* nur wenn Teilnehmer ID's vorhanden sind *)
		debug_index := IP_C.FIFO.NR;
		debug_ID := BYTE_TO_INT(IP_C.FIFO.X[debug_index]);
	END_IF;
END_IF;*)
(* -----------------------------------------------------------------------------*)

(* read system time *)
tx := T_PLC_MS();

IF IP_C.C_PORT = 0 THEN
	IP_C.C_PORT := PORT; (* uebergebenen PORT durch parametrierten PORT ersetzen *)
END_IF;
IF IP_C.C_IP = 0 AND IP_C.C_MODE < 4 THEN
	IP_C.C_IP := IP; (* uebergebene IP durch paramtrierte IP ersetzen *)
END_IF;

new_connection := c_ip <> IP_C.C_IP OR c_mode <> IP_C.C_MODE OR c_port <> IP_C.C_PORT; (* neue Verbindungs erwünscht ? *)
c_enable := IP_C.C_ENABLE AND NOT new_connection;

IF IP_C.C_ENABLE AND IP_C.ERROR = 0 AND state = STOP THEN (* Freigabe,kein Fehler,kein Socket offen *)
	c_ip   := IP_C.C_IP;
	c_mode := IP_C.C_MODE;
	c_port := IP_C.C_PORT;
	c_ip_str := IP4_TO_STRING(c_ip);
	udp_mode := C_MODE.0; (* Mode 1,3,5 = udp *)

	error_time := TIME_TO_DWORD(MAX(T#200ms,TIME_OUT));
	IP_C.TIME_RESET := TRUE; (* Alle Timer ruecksetzen *)
	r_max_size := SIZEOF(R_BUF.BUFFER);
	s_max_size := SIZEOF(S_BUF.BUFFER);

	IF udp_mode THEN (* Mode: 1,3,5 = UDP CLIENT/SERVER *)
		state := UDP_INIT;
	ELSIF c_mode = 0 THEN (* Mode: 0 = TCP CLIENT *)
		state := TC_INIT;
	ELSE
		state := TS_INIT; (* Mode: 2,4 = TCP SERVER *)
	END_IF;

	IF c_mode < 5 THEN (* Empfänger-IP vorgeben *)
		s_ip_str := c_ip_str;
		s_ip_exist := TRUE;
	ELSE
		s_ip_str := '';
		s_ip_exist := FALSE;
	END_IF;

	(* ---------------------- Debug-Message ----------------------------*)
	(*IF _debug_enable THEN
		LOG_CL.NEW_MSG := 'IP_CON: MODE ~1 / IP ~2 / PORT ~3 /ID ~6';
		LOG_CL.PRINTF[1] := BYTE_TO_STRING(C_MODE);
		LOG_CL.PRINTF[2] := IP4_TO_STRING(c_ip);
		LOG_CL.PRINTF[3] := WORD_TO_STRING(c_port);
		LOG_CL.PRINTF[6] := INT_TO_STRING(debug_ID);
		LOG_MSG();
	END_IF;*)
	(* -----------------------------------------------------------------------------*)

END_IF;

(* ---------------------- Debug-Message ----------------------------*)
(*IF  _debug_enable THEN
	IF state <> state_last THEN
		LOG_CL.NEW_MSG := 'IP_STEP ~1 -IP_ID ~6';
		LOG_CL.PRINTF[1] := BYTE_TO_STRING(state);
		LOG_CL.PRINTF[6] := INT_TO_STRING(debug_ID);
		LOG_MSG();
		state_last := state;
	END_IF;
END_IF;*)
(* -----------------------------------------------------------------------------*)

IF IP_C.TIME_RESET THEN (* Alle Timer ruecksetzen *)
	IP_C.TIME_RESET := FALSE; (* Reset rücksetzen *)
	c_time := tx; (* Connect Timer ruecksetzen *)
	s_time := tx; (* Send Timer ruecksetzen *)
	r_time := tx; (* Receive Timer ruecksetzen *)

	c_status := BYTE#0; (* letzten Connect Fehler rücksetzen *)
	s_status := BYTE#0; (* letzten Send Fehler rücksetzen *)
	r_status := BYTE#0; (* letzten Receive Fehler rücksetzen *)
END_IF;

(* ---------------------------------------------- *)

CASE state OF

UDP_INIT: (* UDP_CLIENT + SERVER *)
	(* 1. bei UDP-Client wird als lokalport 0 vorgegeben, damit das System automatisch einen freien lokalen Port sucht
	    2. bei UDP Server muss der gewüschte lokalport verwendet werden *)

	fbCreate(bExecute := FALSE);
	fbCreate(	bExecute := TRUE , sSrvNetId := '', sLocalHost := '', nLocalPort := SEL(c_mode = 1,c_port,0) , tTimeOut := TIME_OUT);
	fbCreate.bExecute := FALSE; (* vorbelegung *)
	state := UDP_INIT_WAIT;

UDP_INIT_WAIT:
	fbCreate();
	IF NOT fbCreate.bBusy THEN
		IF NOT fbCreate.bError THEN
			socket := fbCreate.hSocket;
			c_ready := TRUE; (* Connected *)
			state := C_WAIT;
		ELSE
			c_status := 1; (* FB_SocketUdpCreate failed *)
			nErrId := fbCreate.nErrId;
			state := C_CLOSE;
		END_IF;
	END_IF;

(* ---------------------------------------------- *)
TC_INIT: (* TCP-CLIENT (AKTIV) *)
	fbConnect(bExecute := FALSE);
	fbConnect(bExecute := TRUE, sSrvNetId := '', sRemoteHost := c_ip_str, nRemotePort := c_port, tTimeout := TIME_OUT);
	fbConnect.bExecute := FALSE; (* vorbelegung *)
	state := TC_CONNECT;

(* ---------------------------------------------- *)
TC_CONNECT:
	IF NOT c_enable OR c_status = 255 THEN (* keine freigabe oder connect timeout *)
		state := C_CLOSE;
	END_IF;

	fbConnect();
	IF NOT fbConnect.bBusy THEN
		IF fbConnect.bError THEN
			nErrID := fbConnect.nErrId;
			state :=TC_INIT; (* Nochmals versuchen *)
		ELSE
			socket := fbConnect.hSocket;
			c_ready := TRUE; (* Connected *)
			state := C_WAIT;
		END_IF;
	END_IF;
(* ---------------------------------------------- *)
TS_INIT: (* TCP-SERVER (PASSIV) *)
	fbListen(bExecute := FALSE);
	fbListen(bExecute := TRUE , sSrvNetId:= '' , sLocalHost:= '' , nLocalPort:= c_port , tTimeout:= TIME_OUT);
	fbListen.bExecute := FALSE;
	state := TS_LISTEN_WAIT;
(* ---------------------------------------------- *)
TS_LISTEN_WAIT:
	fbListen();
	IF NOT fbListen.bBusy THEN
		IF fbListen.bError THEN
			c_status := 3; (* FB_SocketListen failed *)
			nErrID := fbListen.nErrId;
			state := C_CLOSE;
		ELSE
			server := fbListen.hListener;
			state := TS_ACCEPT;
		END_IF;
	END_IF;
(* ---------------------------------------------- *)
TS_ACCEPT:
	fbAccept(bExecute := FALSE);
	fbAccept(bExecute := TRUE, sSrvNetId := '', hListener := server, tTimeout := TIME_OUT);
	fbAccept.bExecute := FALSE;
	state := TS_ACCEPT_WAIT;
(* ---------------------------------------------- *)
TS_ACCEPT_WAIT:
	fbAccept();
	IF NOT fbAccept.bBusy THEN

		state := TS_ACCEPT; (* vorbelegung  *)

		IF fbAccept.bError THEN
			c_status := 4; (* FB_SocketAccept failed *)
			nErrID := fbAccept.nErrId;
			state := C_CLOSE;
		ELSE (* no error *)
			IF fbAccept.bAccepted THEN
				socket := fbAccept.hSocket;
				IF socket.remoteAddr.sAddr  <> c_ip_str AND c_mode <> 4 THEN
					state := C_CLOSE; (* Remote ablehnen - Verbindung beenden *)
				ELSE
					state := C_WAIT;
					c_ready := TRUE; (* Connected *)
				END_IF;
			END_IF; (* fbAccept.bAccepted *)
		END_IF; (* NOT fbAccept.bError *)
	END_IF; (*  NOT fbAccept.bBusy *)
(* ---------------------------------------------- *)
C_CLOSE:
	c_ready := FALSE;
	IF socket.handle > 0 THEN
		fbClose(bExecute := FALSE );
		fbClose(bExecute := TRUE, sSrvNetId := '',	hSocket := socket);
		fbClose.bExecute := FALSE;
		state := C_CLOSE_WAIT;
	ELSE
		state:= C_CLOSE2;
	END_IF;

C_CLOSE_WAIT:
	fbClose();
	IF NOT fbClose.bBusy THEN
		socket := TCPADS_NULL_HSOCKET; (* Socket rücksetzen *)
		nErrId:= SEL(fbClose.bError,0,fbClose.nErrId);
		state:= C_CLOSE2;
	END_IF;

C_CLOSE2:
	IF server.handle > 0 THEN
		fbClose(bExecute := FALSE );
		fbClose(bExecute := TRUE, sSrvNetId := '',	hSocket := server);
		fbClose.bExecute := FALSE;
		state := C_CLOSE_WAIT2;
	ELSE
		state:= STOP;
	END_IF;

C_CLOSE_WAIT2:
	fbClose();
	IF NOT fbClose.bBusy THEN
		server := TCPADS_NULL_HSOCKET; (* Socket rücksetzen *)
		nErrId:= SEL(fbClose.bError,0,fbClose.nErrId);
		state:= STOP;
	END_IF;

(* ---------------------------------------------- *)

C_WAIT: (* Warten auf Anforderung für Beenden *)
	IF NOT c_enable OR NOT c_ready THEN
		state:= C_CLOSE;
	ELSIF S_BUF.SIZE > 0 AND IP_C.MAILBOX[2] = 0 AND s_ip_exist THEN
		state:= C_SND;
	ELSIF IP_C.MAILBOX[3] = 0 THEN
		state:= C_REC;
	END_IF;

(* ---------------------------------------------- *)

C_REC: (* Daten empfangen *)
	IF R_BUF.SIZE >= INT_TO_UINT(r_max_size) THEN
		R_BUF.SIZE := UINT#0;
		r_status := 254; (* Empfangsbuffer wegen Überlauf rückgesetzt *)
	END_IF;

	r_offset := SEL(udp_mode,UINT_TO_INT(R_BUF.SIZE),0);
	r_count := r_max_size - r_offset;
	bytes_received := 0;

	IF udp_mode THEN
		fbReceiveFrom(bExecute := FALSE );
		fbReceiveFrom(bExecute:= TRUE, sSrvNetId := '', hSocket:= socket, cbLen := r_count, pDest:= ADR(R_BUF.BUFFER), tTimeout:= TIME_OUT);
		fbReceiveFrom.bExecute := FALSE; (* Vorbelegung *)
	ELSE
		fbReceive(bExecute:= FALSE);
		fbReceive(bExecute:= TRUE, sSrvNetId := '' , hSocket:= socket , cbLen:= r_count, pDest:= ADR(R_BUF.BUFFER[r_offset]) , tTimeout:= TIME_OUT);
		fbReceive.bExecute:= FALSE;
	END_IF;
	state := C_REC_WAIT;

C_REC_WAIT:
	IF udp_mode THEN
		fbReceiveFrom(); (* UDP Mode *)
		IF NOT fbReceiveFrom.bBusy THEN
			IF NOT fbReceiveFrom.bError THEN
				IF fbReceiveFrom.nRecBytes > 0 THEN
					IF c_mode <> BYTE#5 AND fbReceiveFrom.sRemoteHost  <> c_ip_str THEN
						R_BUF.SIZE := UINT#0;
					ELSE
						bytes_received := fbReceiveFrom.nRecBytes;
						IF NOT s_ip_exist THEN
							s_ip_str := fbReceiveFrom.sRemoteHost;
							s_ip_exist := TRUE;
						END_IF;
					END_IF;
				END_IF;
				state := C_WAIT;
			ELSIF fbReceiveFrom.nErrId = 16#80072746 THEN (* Verbindung vom Remote beendet *)
				c_status := 253;
				c_ready := FALSE;
				state := C_WAIT;
			ELSE
				nErrId := fbReceiveFrom.nErrId;
				state := C_WAIT;
			END_IF;
		END_IF;
	ELSE
		fbReceive(); (* TCP Mode *)
		IF NOT fbReceive.bBusy THEN
			IF NOT fbReceive.bError THEN
				IF fbReceive.nRecBytes > 0 THEN
					bytes_received := fbReceive.nRecBytes;
				END_IF;
			ELSIF fbReceive.nErrId = 16#8004 THEN (* Verbindung vom Remote beendet *)
				c_status := 253;
				c_ready := FALSE;
			ELSE
				nErrId := fbReceive.nErrId;
			END_IF;
			state := C_WAIT;
		END_IF;
	END_IF;

	IF bytes_received > 0 THEN
		r_time := tx; (* Receive Timer ruecksetzen *)
		R_BUF.SIZE := INT_TO_UINT(r_offset + DINT_TO_UINT(bytes_received)); (* aktuelle buffersize eintragen *)
		IP_C.MAILBOX[1] := IP_C.MAILBOX[1] + 1; (* Receive Info *)
		IF IP_C.MAILBOX[1] = 0 THEN IP_C.MAILBOX[1] := 1; END_IF;
		(* ---------------------- Debug-Message ----------------------------*)
		(*IF _debug_enable THEN
			LOG_CL.NEW_MSG := 'IP_REC DATA: POS: ~1 : SIZE: ~2 TOTAL ~3 -IP_ID ~6';
			LOG_CL.PRINTF[1] := INT_TO_STRING(r_offset);
			LOG_CL.PRINTF[2] := INT_TO_STRING(r_count);
			LOG_CL.PRINTF[3] := UINT_TO_STRING(R_BUF.SIZE);
			LOG_CL.PRINTF[6] := INT_TO_STRING(debug_ID);
			LOG_MSG();
		END_IF;*)
		(* -----------------------------------------------------------------------------*)
	END_IF;

(* ---------------------------------------------- *)
C_SND:
	IF S_BUF.SIZE > 0 THEN
		IF c_ready AND c_enable THEN
			IF NOT s_active THEN
				s_total := LIMIT(0,UINT_TO_INT(S_BUF.SIZE),r_max_size); (* Gesamtanzahl an Bytes limitieren und uebergeben *)
				s_cur_pos  := 0;
				s_cur_size := 0;
				s_active := TRUE; (* Sende-Betrieb aktivieren *)
			END_IF;

			s_cur_pos := s_cur_pos + s_cur_size; (* neue Sende-Datenposition bestimmen *)
			IF s_total > s_cur_pos THEN (* weitere Daten zum senden vorhanden ? *)
				s_cur_size := s_total - s_cur_pos;
				s_cur_size := LIMIT(0, s_cur_size, s_max_size); (* Telegrammlänge begrenzen *)
				s_time := tx; (* Send Timer ruecksetzen *)
				r_time := tx; (* Receive Timer ruecksetzen *)
				state := C_SND_WAIT1;
			ELSE (* keine weitere Sendedaten vorhanden -> Senden beenden *)
				s_active := FALSE;
				S_BUF.SIZE := 0;
				state := C_WAIT;
			END_IF;
		END_IF;
	END_IF;

C_SND_WAIT1:
	IF udp_mode THEN
		fbSendTo(bExecute := FALSE );
		fbSendTo(bExecute := TRUE, sSrvNetId := '', hSocket := socket , cbLen := s_cur_size, pSrc := ADR(S_BUF.BUFFER[s_cur_pos]), sRemoteHost := s_ip_str, nRemotePort := c_port, tTimeout:= TIME_OUT);
		fbSendTo.bExecute := FALSE;
	ELSE
		fbSend(bExecute := FALSE);
		fbSend(bExecute := TRUE, sSrvNetId := '', hSocket := socket , cbLen:= s_cur_size, pSrc:=ADR(S_BUF.BUFFER[s_cur_pos]), tTimeout:= TIME_OUT);
		fbSend.bExecute := FALSE;
	END_IF;
	state := C_SND_WAIT2;

C_SND_WAIT2:
	IF udp_mode THEN
		fbSendTo();
		Send_Busy := fbSendTo.bBusy;
		Send_Error := fbSendTo.bError;
		Send_ErrId := fbSendTo.nErrId;
	ELSE
		fbSend();
		Send_Busy := fbSend.bBusy;
		Send_Error := fbSend.bError;
		Send_ErrId := fbSend.nErrId;
	END_IF;

	IF NOT Send_Busy THEN
		IF NOT Send_Error THEN
			(* ---------------------- Debug-Message ----------------------------*)
			(*IF _debug_enable THEN
				LOG_CL.NEW_MSG := 'IP_SEN SEND_COUNT ~1 -IP_ID ~6';
				LOG_CL.PRINTF[1] := DINT_TO_STRING(s_cur_size);
				LOG_CL.PRINTF[6] := INT_TO_STRING(debug_ID);
				LOG_MSG();
			END_IF;*)
			(* -----------------------------------------------------------------------------*)
			state := C_SND;
		ELSE
			nErrId := Send_ErrId;
			state := C_WAIT;
			(* ---------------------- Debug-Message ----------------------------*)
			(*IF _debug_enable THEN
				LOG_CL.NEW_MSG := 'IP_SEN SEND ERROR ~1 -IP_ID ~6';
				LOG_CL.PRINTF[1] := UDINT_TO_STRING(nErrId);
				LOG_CL.PRINTF[6] := INT_TO_STRING(debug_ID);
				LOG_MSG();
			END_IF;*)
			(* -----------------------------------------------------------------------------*)
		END_IF;
	END_IF;

END_CASE;

(* ---------------------------------------------- *)

IF c_ready THEN
	IF NOT c_ready_old THEN (* Verbindung aufgebaut - positive Flanke erkannt *)
		IP_C.C_STATE := 254;
		IP_C.TIME_RESET := TRUE; (* Alle Timer ruecksetzen *)
		(* ---------------------- Debug-Message ----------------------------*)
		(*IF _debug_enable THEN
			LOG_CL.NEW_MSG := 'IP_CON: CONNECTED -IP_ID ~6';
			LOG_CL.PRINTF[6] := INT_TO_STRING(debug_ID);
			LOG_MSG();
		END_IF;*)
		(* -----------------------------------------------------------------------------*)
	ELSE
		IP_C.C_STATE := 255; (* Verbindung ist aufgebaut *)
	END_IF;
ELSE
	IF c_ready_old THEN (* Verbindung abgebaut - negative Flanke erkannt *)
		IP_C.C_STATE := 1;
		IP_C.MAILBOX[1] := 0; (* Receive Info rücksetzen *)
		IP_C.MAILBOX[2] := 0; (* Send-Pause rücksetzen *)
		IP_C.MAILBOX[3] := 0; (* Receive-Pause rücksetzen *)
		IF NOT new_connection THEN
			s_active := FALSE; (* Sendeaktivitäten stoppen *)
			S_BUF.SIZE := 0; (* Sendelänge löschen *)
			(* IP_C.TIME_RESET := TRUE; *) (* Alle Timer ruecksetzen *)
		END_IF;
		(* ---------------------- Debug-Message ----------------------------*)
		(*IF _debug_enable THEN
			LOG_CL.NEW_MSG := 'IP_CON: DISCONNECTED';
			LOG_MSG();
		END_IF;*)
		(* -----------------------------------------------------------------------------*)

	ELSE
		IP_C.C_STATE := 0; (* Verbindung ist abgebaut *)
	END_IF;
END_IF;

c_ready_old := c_ready;

(* ---------------------------------------------- *)

IF IP_C.R_OBSERVE = FALSE OR s_active THEN
    r_time := tx;
END_IF;

IF c_status = 0 AND tx - c_time > error_time AND c_enable AND NOT c_ready AND c_mode < 2 THEN (* Connect Timeout *)
	c_status := 255; (* Timeout-Fehler ausgeben *)
END_IF;
IF s_status = 0 AND tx - s_time > error_time AND s_active THEN (* Send Timeout *)
	s_status := 255; (* Timeout-Fehler ausgeben *)
END_IF;
IF r_status = 0 AND tx - r_time > error_time AND c_ready AND IP_C.R_OBSERVE THEN (* Receive Timeout *)
	r_status := 255; (* Timeout-Fehler ausgeben *)
END_IF;

IP_C.ERROR := DWORD_OF_BYTE(c_status,s_status,r_status,0);

(* ---------------------- Debug-Message ----------------------------*)
(*IF  _debug_enable THEN
	IF (IP_C.ERROR <> debug_lasterror) THEN
		LOG_CL.NEW_MSG := 'IP_ERROR ~1 -IP_ID ~6';
		LOG_CL.PRINTF[1] := DWORD_TO_STRING(IP_C.ERROR);
		LOG_CL.PRINTF[6] := INT_TO_STRING(debug_ID);
		LOG_MSG();

		debug_lasterror := IP_C.ERROR;
		debug_last_id := debug_ID;
	END_IF;
END_IF;*)
(* -----------------------------------------------------------------------------*)

(* revision history
ks	18. oct. 2008	rev 1.0
	original version
ks	05. jan. 2009	rev 1.1
	zusätzlichen Parameter "Port" hinzugefügt, und Code bei Verbindungsaufbau angepasst
ks	28. feb. 2009	rev 1.2
	connect code angepasst und verkürzung der zyklen bei Send
ks	20. oct. 2009	rev 1.3
	network_buffer basis 0
ks	06. dec. 2009	rev 1.4
	receive_count MAILBOX[1]
ks	10. nov. 2010	rev 1.5
	send_pause MAILBOX[2] and receive_pause MAILBOX[3] 
ks	07. feb. 2011	rev 1.6
	Fehlercode 253 bei Remote-Verbindungsabbruch 
ks	30. may. 2011	rev 1.7
	Fehler bei Empfangsüberwachung
ks	26. july. 2011	rev 1.8
	Error-Reset, diverse optimierungen 
*)

END_FUNCTION_BLOCK

// ---- beckhoff_network/POUs/NETWORK/MB_SERVER.TcPOU
FUNCTION_BLOCK MB_SERVER
VAR_IN_OUT
	IP_C : IP_C;
	S_BUF : NETWORK_BUFFER_SHORT;
	R_BUF : NETWORK_BUFFER_SHORT;
	VMAP : ARRAY [1..10] OF VMAP_DATA;
	DATA : ARRAY [0..255] OF WORD;
END_VAR
VAR_INPUT
	DATA_SIZE : INT;
	ENABLE : BOOL;
	UDP : BOOL;
END_VAR
VAR_OUTPUT
	ERROR : DWORD;
END_VAR
VAR
	MB_VMAP : MB_VMAP;
	adr1 : INT;
	adr2 : INT;
	points : INT;
	points2 : INT;
	coils : BYTE;
	mask : BYTE;
	idx1 : INT;
	idx2 : INT;
	bit_pos : INT;
	count : INT;
	fc : INT;
	i : INT;
	state : INT;
	ip_state : BYTE;
	ip_id : BYTE;
	IP_FIFO : IP_FIFO;
	w_tmp : WORD;
	last_cycle : TIME;
	tx : TIME;
	t : TON;
	ip_error : BOOL;
END_VAR

(*

version 1.3		17. may. 2011
programmer 		ks
tested by			ks

MB_SERVER ermöglicht das Lesen/Schreiben von Daten durch ein Remote-Device mittels Modbus over Ethernet (OpenModbus)

*)

(* read system time *)
tx := DWORD_TO_TIME(T_PLC_MS());

FOR i := 1 TO 10 DO
	IF VMAP[i].TIME_OUT > T#0s THEN
		VMAP[i].TIME_OUT := VMAP[i].TIME_OUT + tx - last_cycle;
	END_IF;
END_FOR;
last_cycle := tx;
ip_error := IP_C.ERROR > DWORD#0;

CASE state OF
00: (* Warten auf Freigabe *)
	IF ENABLE THEN
		state := 10;
		ip_state := BYTE#1; (* Anmelden *)
	END_IF;

10: (* Bei IP_Control anmelden und auf freigabe warten *)
	IF ip_state = BYTE#3 THEN

		(* IP Datenverkehr einrichten *)
		IP_C.C_PORT := WORD#0; (* Port von IP_CONTROL verwenden *)
		IP_C.C_IP := DWORD#0; (* IP von IP_CONTROL verwenden *)
		IP_C.C_MODE := SEL(UDP,BYTE#4,BYTE#5); (* Mode: 4=TCP+PASSIV+PORT , 5=UDP+PASSIV+PORT *)
		IP_C.TIME_RESET := TRUE; (* Zeitueberwachung rücksetzen *)
		IP_C.C_ENABLE := TRUE; (* Verbindungsaufbau freigeben *)
		IP_C.R_OBSERVE := FALSE; (* keine Empfangsueberwachung *)
		state := 20;
	END_IF;

20:	IF NOT ip_error THEN
		IF S_BUF.SIZE = UINT#0 AND R_BUF.SIZE > UINT#6 THEN	(* Datensenden nicht aktiv und Daten wurden empfangen *)
			IF  R_BUF.SIZE = WORD_TO_UINT(WORD_OF_BYTE(R_BUF.BUFFER[4],R_BUF.BUFFER[5])) + UINT#6 THEN (* gültige Datenlänge *)
				ERROR := DWORD#00; (* Error löschen *)
	
				(* Header kopieren *)
				FOR i := 0 TO 13 DO
					S_BUF.BUFFER[i] := R_BUF.BUFFER[i];
				END_FOR;
				fc := BYTE_TO_INT(R_BUF.BUFFER[7]);
				adr1 := WORD_TO_INT(WORD_OF_BYTE(R_BUF.BUFFER[8],R_BUF.BUFFER[9]));
				points := WORD_TO_INT(WORD_OF_BYTE(R_BUF.BUFFER[10],R_BUF.BUFFER[11]));
	
				(* Virtual Address *)
				MB_VMAP(VMAP:=VMAP,FC:=fc,V_ADR:=adr1,V_CNT:=points,SIZE:=DATA_SIZE);
				adr1:=MB_VMAP.P_ADR;
				bit_pos:=MB_VMAP.P_BIT;
				ERROR:=BYTE_TO_DWORD(MB_VMAP.ERROR);
	
				IF ERROR = DWORD#0 THEN
					CASE fc OF
					(*---------------------------------------------*)
					1..2 : (* Read Coil Status / Read Input Status *)
						count := 9; (* erstes Datenbyte *)
						coils := BYTE#0;
						mask := BYTE#1;
						FOR i := 1 TO points DO
							IF mask = BYTE#0 THEN
								mask := BYTE#1;
								S_BUF.BUFFER[count] := coils;
								coils := BYTE#0;
								count := count + 1;
							END_IF;
							IF (DATA[adr1] AND SHL(WORD#1,bit_pos)) > WORD#0 THEN
								coils := coils OR mask;
							END_IF;
	
							bit_Pos := bit_Pos + 1;
							IF bit_pos > 15 THEN
								ADR1 := ADR1 + 1;
								bit_pos := 0;
							END_IF;
	
							mask := SHL(mask,1);
						END_FOR;
						S_BUF.BUFFER[Count] := coils;
	
						S_BUF.BUFFER[8] := INT_TO_BYTE(count - 8); (* Bytecount *)
						S_BUF.SIZE := INT_TO_UINT(count + 1);
	
					(*--------------------------------------------------*)
					3..4 : (* Read Holding Registers / Read Input Registers *)
						idx1 := 07;
						count := adr1 + points - 1;
						FOR i := adr1 TO count DO
							idx1 := idx1 + 2;
							idx2 := idx1 + 1; (* zweiter index für pcworx notwendig ! *)
							w_tmp := DATA[i];
							S_BUF.BUFFER[idx1] := WORD_TO_BYTE(SHR(w_tmp,8));
							S_BUF.BUFFER[idx2] := WORD_TO_BYTE(w_tmp);
						END_FOR;
						S_BUF.BUFFER[8] := SHL(INT_TO_BYTE(points),1); (* Anzahl Register in Bytes *)
						S_BUF.SIZE := INT_TO_UINT(idx2 + 1);
					(*--------------------------------------------------*)
					5 : (* Force Single Coil *)
						DATA[adr1]:=BIT_LOAD_W(DATA[adr1],R_BUF.BUFFER[10] > BYTE#0,bit_pos);
						S_BUF.SIZE := UINT#12;
					(*--------------------------------------------------*)
					6 : (* Preset Single Register *)
						DATA[adr1] := WORD_OF_BYTE(R_BUF.BUFFER[10],R_BUF.BUFFER[11]);
						S_BUF.SIZE := UINT#12;
					(*--------------------------------------------------*)
					15 : (* Force Multible Coils *)
						mask := BYTE#1;
						idx1 := 13;
						FOR i := 1 TO points DO
							DATA[adr1]:=BIT_LOAD_W(DATA[adr1],(R_BUF.BUFFER[idx1] AND mask) > BYTE#0,bit_pos);
							bit_pos := bit_pos + 1;
							IF bit_pos > 15 THEN
								adr1:= adr1 + 1;
								bit_pos := 0;
							END_IF;
							mask := ROL(mask,1);
							IF mask = BYTE#1 THEN
								idx1 := idx1 +1;
							END_IF;
						END_FOR;
						S_BUF.SIZE := UINT#12;
					(*--------------------------------------------------*)
					16 : (* Preset Multiple Registers	*)
						idx1 := 11;
						count := adr1 + points - 1;
						FOR i := adr1 TO Count DO
							idx1 := idx1 + 2;
	 						idx2 := idx1 + 1;
							Data[i] := WORD_OF_BYTE(R_BUF.BUFFER[idx1],R_BUF.BUFFER[idx2]);
						END_FOR;
						S_BUF.SIZE := UINT#12;
					(*--------------------------------------------------*)
					22 : (* Mask Write Register *)
						w_tmp := WORD_OF_BYTE(R_BUF.BUFFER[10],R_BUF.BUFFER[11]); (* and mask *)
						DATA[adr1] := (DATA[adr1] AND w_tmp) OR (WORD_OF_BYTE(R_BUF.BUFFER[12],R_BUF.BUFFER[13]) AND (NOT w_tmp));
						S_BUF.SIZE := UINT#14;
					(*--------------------------------------------------*)
					23 : (* Read / Write Registers	*)
						(*--- Write-Register -----------------------------------*)
						adr2 := WORD_TO_INT(WORD_OF_BYTE(R_BUF.BUFFER[12],R_BUF.BUFFER[13]));
						points2 := WORD_TO_INT(WORD_OF_BYTE(R_BUF.BUFFER[14],R_BUF.BUFFER[15]));
	
						(* Virtual Address Write Register *)
						MB_VMAP(VMAP:=VMAP,FC:=16,V_ADR:=adr2,V_CNT:=points2,SIZE:=DATA_SIZE);
						adr2:=MB_VMAP.P_ADR;
						ERROR:=BYTE_TO_DWORD(MB_VMAP.ERROR);
	
						IF ERROR = DWORD#0 THEN
							idx1 := 15;
							count := adr2 + points2 - 1;
							FOR i := adr2 TO count DO
								idx1 := idx1 + 2;
	 							idx2 := idx1 + 1; (* zweiter index für pcworx notwendig ! *)
								Data[i] := WORD_OF_BYTE(R_BUF.BUFFER[idx1],R_BUF.BUFFER[idx2]);
							END_FOR;
	
							(*--- Read-Register -----------------------------------*)
							idx1 := 07;
							count := adr1 + points - 1;
							FOR i := adr1 TO count DO
								idx1 := idx1 + 2;
								idx2 := idx1 + 1; (* zweiter index für pcworx notwendig ! *)
								w_tmp := DATA[i];
								S_BUF.BUFFER[idx1] := WORD_TO_BYTE(SHR(w_tmp,8));
								S_BUF.BUFFER[idx2] := WORD_TO_BYTE(w_tmp);
							END_FOR;
							S_BUF.BUFFER[8] := SHL(INT_TO_BYTE(points),1); (* Anzahl Register in Bytes *)
							S_BUF.SIZE := INT_TO_UINT(idx2 + 1);
	
						END_IF;
	
					(*--------------------------------------------------*)
					ELSE
						ERROR := DWORD#01; (* ILLEGAL FUNCTION *)
					END_CASE;
				END_IF;
			END_IF;
	
			IF ERROR > DWORD#0 THEN
				S_BUF.BUFFER[7] := S_BUF.BUFFER[7] OR BYTE#2#1000_0000; (* Fehlerbit setzen *)
				S_BUF.BUFFER[8] := DWORD_TO_BYTE(ERROR);
				S_BUF.SIZE := UINT#9;
			END_IF;
	
			S_BUF.BUFFER[4] := BYTE#0; (* high Byte *)
			S_BUF.BUFFER[5] := UINT_TO_BYTE(S_BUF.SIZE - UINT#6); (* Längenfeld eintragen - nur low byte *)
	
		END_IF;
	ELSE
		ERROR := IP_C.ERROR;
	END_IF;

	t(IN:= ip_error, PT:=T#5s);
	IF t.Q THEN
		IP_C.TIME_RESET := TRUE; (* Error Reset *)
	END_IF;



	R_BUF.SIZE := UINT#0; (* Empfangsdaten zerstören *)

	IF ENABLE = FALSE THEN
	    ip_state := BYTE#4; (* Abmelden *)
		state := 00;
	END_IF;
END_CASE;

(* IP_FIFO *)
IP_FIFO(FIFO:=IP_C.FIFO,STATE:=ip_state,ID:=ip_id);

(* revision history
ks	05. jan. 2009	rev 1.0
	original version

ks	28. jan. 2009	rev 1.1
	network_buffer_short verwendet  

ks	20. oct. 2009	rev 1.2
	change lokal-var adr to adr1,Networkbuffer und Buffer-funktionen auf Basis 0

ks	17. may. 2011	rev 1.3
	automatischer re-connect
*)

END_FUNCTION_BLOCK

// ---- beckhoff_network/POUs/NETWORK/MB_VMAP.TcPOU
FUNCTION_BLOCK MB_VMAP
VAR_IN_OUT
	VMAP :  ARRAY [1..10] OF VMAP_DATA;
END_VAR
VAR_INPUT
	FC : INT;
	V_ADR : INT;
	V_CNT : INT;
	SIZE : INT;
END_VAR
VAR_OUTPUT
	P_ADR : INT;
	P_BIT : INT;
	ERROR : BYTE;
END_VAR
VAR
	i : INT;
	vopt : DWORD;
	vadr : INT;
	padr : INT;
	mask : DWORD;
	vsize : INT;
	w_tmp : WORD;
	i_tmp : INT;
	init : BOOL;
END_VAR

(*
version 1.1		20. oct. 2009
programmer 		ks
tested by		ks

MB_VMAP Virtuelles Adress-Mapping für MB_SERVER
*)

IF init = FALSE THEN
	init := TRUE;
	IF VMAP[1].FC = DWORD#0 THEN
		VMAP[1].FC := DWORD#16#FFFF_FFFF;
		VMAP[1].V_ADR := 0;
		VMAP[1].V_SIZE := 256;
		VMAP[1].P_ADR := 0;
	END_IF;
END_IF;

ERROR := BYTE#02; (* ILLEGAL DATA ADDRESS *)
mask := SHL(DWORD#1,FC);

IF (mask AND DWORD#2#00000000_01000000_00000000_01100000) <> DWORD#0 THEN (* FC 5,6,22 *)
	V_CNT := 1;
ELSIF V_CNT = 0 THEN
	RETURN;
END_IF;

FOR i := 1 TO 10 DO
	vopt := VMAP[i].FC; 
	IF (vopt AND mask) <> DWORD#0 THEN
		vadr := VMAP[i].V_ADR;
		vsize := VMAP[i].V_SIZE;
		padr := VMAP[i].P_ADR;

		IF (mask AND DWORD#2#00000000_00000000_10000000_00100110) <> DWORD#0 THEN (* FC 1,2,5,15 für Bit-Access *)
			i_tmp := WORD_TO_INT(SHR(INT_TO_WORD(V_ADR + V_CNT -1),4))+1;
			IF i_tmp <= SIZE AND i_tmp <= vsize THEN
				w_tmp := INT_TO_WORD(V_ADR);
				P_ADR := WORD_TO_INT(SHR(w_tmp,4)) + padr; 
				P_BIT := WORD_TO_INT(w_tmp AND WORD#16#000F);
				ERROR := BYTE#0;
				EXIT;
			END_IF;
		ELSIF (mask AND DWORD#2#00000000_11000001_00000000_01011000) <> DWORD#0 THEN (* FC 3,4,6,16,22,23 für Register-Access *)
			IF V_ADR >= vadr AND V_ADR + V_CNT <= vadr + vsize THEN (* gültiger virtueller bereich *)
				P_ADR := V_ADR - vadr + padr; (* reale Adresse berechnen *)
				IF P_ADR + V_CNT <= SIZE THEN (* bereichsueberschreitung ? *)
					ERROR := BYTE#0;
					EXIT;
				END_IF;
			END_IF;
		ELSE
			ERROR := BYTE#01; (* ILLEGAL FUNCTION *)
			RETURN;
		END_IF;
	END_IF;
END_FOR;

IF ERROR = BYTE#0 THEN
	IF (mask AND DWORD#2#00000000_11000001_10000000_01100000) <> DWORD#0 THEN (* FC 5,6,15,16,22,23 Schreib-zugriff *)
		VMAP[i].TIME_OUT := T#1ms;
	END_IF;
END_IF;

(* revision history
ks	05. jan. 2009	rev 1.0
	original version

ks	20. oct. 2009	rev 1.1
	fehlerkorrektur in bitmaske

*)

END_FUNCTION_BLOCK

// ---- oscat_basic/POUs/Logic/gate logic/BIT_LOAD_W.TcPOU
FUNCTION BIT_LOAD_W : WORD
VAR_INPUT
	IN : WORD;
	VAL : BOOL;
	POS : INT;
END_VAR
VAR CONSTANT
	dat : WORD := 1;
END_VAR

(*
version 1.1	16. mar 2008
programmer 	hugo
tested by	tobias

this function loads a bit into a Word at position pos.
 *)

IF val THEN
	BIT_LOAD_W := in OR SHL(dat,pos);
ELSE
	BIT_LOAD_W := in AND (NOT SHL(dat,pos));
END_IF;


(* revision history
hm	29. feb 2008	rev 1.0
	original version

hm	16. mar 2008	rev 1.1
	change input bit to val for compatibility reasons
*)

END_FUNCTION

// ---- beckhoff_network/POUs/DEMO/MD5_CRAM_AUTH_DEMO.TcPOU
PROGRAM MD5_CRAM_AUTH_DEMO
VAR
	run: BOOL := TRUE;
	timestamp : STRING(64) := 'PDQwMzYuMTA3NjMyNDM4MUBndWlsZGVuc3Rlcm4uemVpdGZvcm0uZGU+';
	password : STRING := 'geheimes_passwort';
	username : STRING := 'benutzer@zeitform.de';
	auth_key : STRING(STRING_LENGTH);
	MD5_CRAM_AUTH: MD5_CRAM_AUTH;
END_VAR

// Beispiel:
MD5_CRAM_AUTH(
    RUN := run,
    USERNAME := username,
    PASSWORD := password,
    B64_TS := timestamp,
    AUTH_KEY := auth_key);

END_PROGRAM

// ---- beckhoff_network/POUs/DEMO/NET_VAR_MASTER_DEMO.TcPOU
PROGRAM NET_VAR_MASTER_DEMO
VAR
	NET_VAR_CONTROL_1: NET_VAR_CONTROL;
	activate: BOOL := TRUE;
	run: BOOL;
	udp: BOOL := TRUE;
	master: BOOL := TRUE;
	remote_port: WORD := 10000;
	scan_time: TIME := T#1s;
	watchdog: TIME := T#2s;
	error: DWORD;
	x: NET_VAR_DATA;

	NET_VAR_BOOL8_1: NET_VAR_BOOL8;
	id_b8: BYTE;
	in_b1: BOOL;
	in_b2: BOOL;
	in_b3: BOOL;
	in_b4: BOOL;
	in_b5: BOOL;
	in_b6: BOOL;
	in_b7: BOOL;
	in_b8: BOOL;
	out_b1: BOOL;
	out_b2: BOOL;
	out_b3: BOOL;
	out_b4: BOOL;
	out_b5: BOOL;
	out_b6: BOOL;
	out_b7: BOOL;
	out_b8: BOOL;

	NET_VAR_STRING_1: NET_VAR_STRING;
	in_s1: STRING(STRING_LENGTH);
	out_s1: STRING(STRING_LENGTH);
	id_s: BYTE;

	NET_VAR_BUFFER_1: NET_VAR_BUFFER;
	id_bu: BYTE;
	BUF_IN : ARRAY [1..64] OF BYTE;
	BUF_OUT : ARRAY [1..64] OF BYTE;

	id_dw: BYTE;
	NET_VAR_DWORD8_1: NET_VAR_DWORD8;
	in_dw1 : DWORD;
	in_dw2 : DWORD;
	in_dw3 : DWORD;
	in_dw4 : DWORD;
	in_dw5 : DWORD;
	in_dw6 : DWORD;
	in_dw7 : DWORD;
	in_dw8 : DWORD;
	out_dw1 : DWORD;
	out_dw2 : DWORD;
	out_dw3 : DWORD;
	out_dw4 : DWORD;
	out_dw5 : DWORD;
	out_dw6 : DWORD;
	out_dw7 : DWORD;
	out_dw8 : DWORD;

	NET_VAR_REAL8_1: NET_VAR_REAL8;
	in_r1 : REAL;
	in_r2 : REAL;
	in_r3 : REAL;
	in_r4 : REAL;
	in_r5 : REAL;
	in_r6 : REAL;
	in_r7 : REAL;
	in_r8 : REAL;
	out_r1 : REAL;
	out_r2 : REAL;
	out_r3 : REAL;
	out_r4 : REAL;
	out_r5 : REAL;
	out_r6 : REAL;
	out_r7 : REAL;
	out_r8 : REAL;
	id_r: BYTE;

	NET_VAR_X8_1: NET_VAR_X8;
	in_x_re1 : REAL;
	in_x_re2 : REAL;
	in_x_di1 : DINT;
	in_x_di2 : DINT;
	in_x_ud1 : UDINT;
	in_x_ud2 : UDINT;
	in_x_dw1 : DWORD;
	in_x_dw2 : DWORD;
	out_x_re1 : REAL;
	out_x_re2 : REAL;
	out_x_di1 : DINT;
	out_x_di2 : DINT;
	out_x_ud1 : UDINT;
	out_x_ud2 : UDINT;
	out_x_dw1 : DWORD;
	out_x_dw2 : DWORD;
	id_x8: BYTE;
END_VAR
VAR // added by the converter: edge detectors and wires of the graphical bodies
    _w1 : ANY;
END_VAR

NET_VAR_DWORD8_1(
    IN1 := in_dw1,
    IN2 := in_dw2,
    IN3 := in_dw3,
    IN4 := in_dw4,
    IN5 := in_dw5,
    IN6 := in_dw6,
    IN7 := in_dw7,
    IN8 := in_dw8,
    X := x); // NET_VAR_DWORD8
out_dw1 := NET_VAR_DWORD8_1.OUT1;
out_dw2 := NET_VAR_DWORD8_1.OUT2;
out_dw3 := NET_VAR_DWORD8_1.OUT3;
out_dw4 := NET_VAR_DWORD8_1.OUT4;
out_dw5 := NET_VAR_DWORD8_1.OUT5;
out_dw6 := NET_VAR_DWORD8_1.OUT6;
out_dw7 := NET_VAR_DWORD8_1.OUT7;
out_dw8 := NET_VAR_DWORD8_1.OUT8;
id_dw := NET_VAR_DWORD8_1.ID;
NET_VAR_REAL8_1(
    IN1 := in_r1,
    IN2 := in_r2,
    IN3 := in_r3,
    IN4 := in_r4,
    IN5 := in_r5,
    IN6 := in_r6,
    IN7 := in_r7,
    IN8 := in_r8,
    X := x); // NET_VAR_REAL8
out_r1 := NET_VAR_REAL8_1.OUT1;
out_r2 := NET_VAR_REAL8_1.OUT2;
out_r3 := NET_VAR_REAL8_1.OUT3;
out_r4 := NET_VAR_REAL8_1.OUT4;
out_r5 := NET_VAR_REAL8_1.OUT5;
out_r6 := NET_VAR_REAL8_1.OUT6;
out_r7 := NET_VAR_REAL8_1.OUT7;
out_r8 := NET_VAR_REAL8_1.OUT8;
id_r := NET_VAR_REAL8_1.ID;
NET_VAR_BOOL8_1(
    IN1 := in_b1,
    IN2 := in_b2,
    IN3 := in_b3,
    IN4 := in_b4,
    IN5 := in_b5,
    IN6 := in_b6,
    IN7 := in_b7,
    IN8 := in_b8,
    X := x); // NET_VAR_BOOL8
out_b1 := NET_VAR_BOOL8_1.OUT1;
out_b2 := NET_VAR_BOOL8_1.OUT2;
out_b3 := NET_VAR_BOOL8_1.OUT3;
out_b4 := NET_VAR_BOOL8_1.OUT4;
out_b5 := NET_VAR_BOOL8_1.OUT5;
out_b6 := NET_VAR_BOOL8_1.OUT6;
out_b7 := NET_VAR_BOOL8_1.OUT7;
out_b8 := NET_VAR_BOOL8_1.OUT8;
id_b8 := NET_VAR_BOOL8_1.ID;
NET_VAR_BUFFER_1(BUF_IN := BUF_IN, BUF_OUT := BUF_OUT, X := x); // NET_VAR_BUFFER
id_bu := NET_VAR_BUFFER_1.ID;
NET_VAR_STRING_1(IN := in_s1, OUT := out_s1, X := x); // NET_VAR_STRING
id_s := NET_VAR_STRING_1.ID;
NET_VAR_X8_1(
    IN_REAL1 := in_x_re1,
    IN_REAL2 := in_x_re2,
    IN_DINT1 := in_x_di1,
    IN_DINT2 := in_x_di2,
    IN_UDINT1 := in_x_ud1,
    IN_UDINT2 := in_x_ud2,
    IN_DWORD1 := in_x_dw1,
    IN_DWORD2 := in_x_dw2,
    X := x); // NET_VAR_X8
out_x_re1 := NET_VAR_X8_1.OUT_REAL1;
out_x_re2 := NET_VAR_X8_1.OUT_REAL2;
out_x_di1 := NET_VAR_X8_1.OUT_DINT1;
out_x_di2 := NET_VAR_X8_1.OUT_DINT2;
out_x_ud1 := NET_VAR_X8_1.OUT_UDINT1;
out_x_ud2 := NET_VAR_X8_1.OUT_UDINT2;
out_x_dw1 := NET_VAR_X8_1.OUT_DWORD1;
out_x_dw2 := NET_VAR_X8_1.OUT_DWORD2;
id_x8 := NET_VAR_X8_1.ID;
_w1 := DWORD_OF_BYTE(192, 168, 178, 50);
NET_VAR_CONTROL_1(
    ACTIVATE := activate,
    MASTER := master,
    UDP := udp,
    REMOTE_IP4 := _w1,
    REMOTE_PORT := remote_port,
    SCAN_TIME := scan_time,
    WATCHDOG := watchdog,
    X := x); // NET_VAR_CONTROL
run := NET_VAR_CONTROL_1.RUN;
error := NET_VAR_CONTROL_1.ERROR;

END_PROGRAM

// ---- beckhoff_network/POUs/NET_VAR/NET_VAR_CONTROL.TcPOU
FUNCTION_BLOCK NET_VAR_CONTROL
VAR_INPUT
	ACTIVATE : BOOL;
	MASTER : BOOL;
	UDP : BOOL;
	REMOTE_IP4 : DWORD;
	REMOTE_PORT : WORD := 10000;
	SCAN_TIME : TIME := T#1s;
	WATCHDOG : TIME := T#2s;
END_VAR
VAR_OUTPUT
	RUN : BOOL;
	ERROR : DWORD;
END_VAR
VAR_IN_OUT
	X : NET_VAR_DATA;
END_VAR
VAR
	IPC : IP_CONTROL;
	IP_C : IP_C; (* IP_Control Verwaltungsstruktur *)
	step : INT;
	activate_last : BOOL;
	tscan : TON;
	reset : BOOL;
END_VAR

(*
version 1.0		15. may. 2011
programmer		ks
tested by			ks

NET_VAR_CONTROL überträgt Daten bidirektional vom Master zum Client
*)

(* Typ
001 = BYTE
002 = WORD
003 = DWORD
004 = BOOL (8x)
005 = REAL
006 = STRING
007 = UINT
008 = INT
009 = DINT
010 = UDINT
013 = DWORD (8x)
015 = REAL (8x)

020 = BUFFER
021 = MIX (REAL,DINT,UDINT,
*)

IF X.ERROR_ID > BYTE#0 THEN (* Schwere Fehler bei Variablenzuordnung vorhanden  !! *)
	X.STATE := BYTE#0;
	ERROR := BYTE_TO_DWORD(X.ERROR_ID);
	X.ERROR_ID := BYTE#0;
	step := 999;
END_IF;

CASE step OF

00:	IF ACTIVATE AND NOT activate_last OR reset THEN

        (*  TCP + MASTER = C_MODE 0 (TCP + ACTIVE + PORT + IP) *)
        (*  UDP + MASTER = C_MODE 1 (UDP + ACTIVE + PORT + IP) *)
        (*  TCP + SLAVE  = C_MODE 2 (TCP + PASSIV + PORT + IP) *)
        (*  UDP + SLAVE  = C_MODE 3 (UDP + PASSIV + PORT + IP) *)
	IF MASTER THEN
		IP_C.C_MODE := BYTE#0;
		step := 100;
	ELSE
		IP_C.C_MODE := BYTE#2;
		step := 200;
	END_IF;
        IF UDP THEN IP_C.C_MODE := IP_C.C_MODE OR BYTE#1; END_IF;
	  	IP_C.C_PORT := REMOTE_PORT; (* Portnummer eintragen *)
	  	IP_C.C_IP := REMOTE_IP4; (* IP eintragen *)
	  	IP_C.TIME_RESET := TRUE; (* Zeitueberwachung rücksetzen *)
	  	IP_C.C_ENABLE := TRUE; (* Verbindungsaufbau freigeben *)
	  	IP_C.R_OBSERVE := TRUE; (* Empfangsueberwachung *)
		X.S_BUF.SIZE := UINT#0;
		X.R_BUF.SIZE := UINT#0;
		X.CYCLE := UDINT#0;
		X.ERROR_ID := BYTE#0;
		reset := FALSE;
	END_IF;

(* ++++++++++++++++++++++++++++++++++++++++++++++ *)

100:IF IP_C.C_STATE > BYTE#127 THEN (* Verbindung vorhanden *)
		X.STATE := BYTE#1; (* Daten sammeln *)
		X.BUF_SIZE := SIZEOF(X.S_BUF.BUFFER);
		X.S_BUF.BUFFER[0] := UDINT_TO_BYTE(X.CYCLE);
		X.INDEX := 1;
		step := 110;
	END_IF;

110:X.STATE := BYTE#0;
	X.S_BUF.SIZE := INT_TO_UINT(X.INDEX); (* Datenlänge eintragen *)
	step := 120;

120:IF X.S_BUF.SIZE = UINT#0 AND X.R_BUF.SIZE >= UINT#1 THEN (* länge der empfangenen Daten prüfen *)
		X.STATE := BYTE#2; (* Daten ausgeben *)
		X.BUF_SIZE := X.R_BUF.SIZE;
		X.INDEX := 1;
		X.ERROR_ID := BYTE#0;
		X.CYCLE := X.CYCLE + UDINT#1;
		ERROR := DWORD#0; (* nach erfolgreichen Zyklus letzten Fehlercode löschen *)
		RUN := TRUE;
		step := 130;
	END_IF;

130:X.STATE := BYTE#0;
	X.R_BUF.SIZE := UINT#0;
	IF NOT ACTIVATE THEN
		step := 999; (* Beenden *)
	ELSIF tscan.Q THEN
		step := 100;
	END_IF;

(* ++++++++++++++++++++++++++++++++++++++++++++++ *)

200:IF X.R_BUF.SIZE >= UINT#1 THEN
		X.STATE := BYTE#2; (* Daten ausgeben *)
		X.BUF_SIZE := X.R_BUF.SIZE;
		X.INDEX := 1;
		step := 210;
	END_IF;

210:X.STATE := BYTE#1; (* Daten sammeln *)
	X.BUF_SIZE := SIZEOF(X.R_BUF.BUFFER);;
	X.S_BUF.BUFFER[0] := X.R_BUF.BUFFER[0]; (* Cycle übernehmen *)
	X.INDEX := 1;
	X.R_BUF.SIZE := UINT#0;
	step := 220;

220:X.STATE := BYTE#0;
	X.S_BUF.SIZE := INT_TO_UINT(X.INDEX); (* Datenlänge eintragen *)
	step := 230;

230:IF X.S_BUF.SIZE = UINT#0 THEN
		ERROR := DWORD#0; (* nach erfolgreichen Zyklus letzten Fehlercode löschen *)
		RUN := TRUE;
		IF NOT ACTIVATE THEN
			step := 999; (* Beenden *)
		ELSE
			step := 200;
		END_IF;
	END_IF;

999:IP_C.C_ENABLE := FALSE; (* Beenden *)
	RUN := FALSE;
	step := 0;

END_CASE;

(* ++++++++++++++++++++++++++++++++++++++++++++++ *)

IPC(IP:= DWORD#0, PORT:= WORD#0 , TIME_OUT:= WATCHDOG, IP_C:= IP_C, S_BUF:= X.S_BUF, R_BUF:= X.R_BUF);

IF IP_C.ERROR > DWORD#0 THEN
	ERROR := IP_C.ERROR;
	RUN := FALSE;
	reset := TRUE;
	step := 0;
END_IF;

ACTIVATE_LAST := ACTIVATE; (* letzten Status sichern zur Flankenerkennung *)
tscan(IN:= step <> 110 ,PT:=SCAN_TIME);

(* revision history
ks	15.may. 2011	rev 1.0
	original version

*)

END_FUNCTION_BLOCK

// ---- beckhoff_network/POUs/NET_VAR/NET_VAR_BOOL8.TcPOU
FUNCTION_BLOCK NET_VAR_BOOL8
VAR_IN_OUT
	X : NET_VAR_DATA;
END_VAR
VAR_INPUT
	IN1 : BOOL;
	IN2 : BOOL;
	IN3 : BOOL;
	IN4 : BOOL;
	IN5 : BOOL;
	IN6 : BOOL;
	IN7 : BOOL;
	IN8 : BOOL;
END_VAR
VAR_OUTPUT
	OUT1 : BOOL;
	OUT2 : BOOL;
	OUT3 : BOOL;
	OUT4 : BOOL;
	OUT5 : BOOL;
	OUT6 : BOOL;
	OUT7 : BOOL;
	OUT8 : BOOL;
	ID : BYTE;
END_VAR
VAR
	init : BOOL;
	index : INT;
	index2 : INT;
	BYTE_TO_BITS : BYTE_TO_BITS;
END_VAR

(*
version 1.0		15. may. 2011
programmer		ks
tested by			ks

NET_VAR_BOOL8 überträgt bidirektional 8 boolsche Werte vom Master zum Client
*)

IF NOT init THEN
	init := TRUE;
	X.ID_MAX := X.ID_MAX + USINT#1;
	ID := USINT_TO_BYTE(X.ID_MAX);
END_IF;

IF X.STATE > BYTE#0 AND X.ERROR_ID = BYTE#0 THEN
	index := X.index; (* PCWORX Workaround *)
	IF INT_TO_UINT(index + 3) > X.BUF_SIZE THEN
		X.ERROR_ID := ID;
	ELSE
		IF X.STATE = BYTE#1 THEN (* Daten schreiben *)
			X.S_BUF.BUFFER[index] := ID; (* ID *)
			index := index + 1;
			X.S_BUF.BUFFER[index] := BYTE#4; (* TYPE BOOL8 *)
			index := index + 1;
			X.S_BUF.BUFFER[index] := BYTE_OF_BIT(IN1,IN2,IN3,IN4,IN5,IN6,IN7,IN8);
			index := index + 1;

		ELSIF X.STATE = BYTE#2 THEN (* Daten lesen *)
			index2 := index + 1; (* PCWORX Workaround *)
			IF X.R_BUF.BUFFER[index] <> ID OR X.R_BUF.BUFFER[index2] <> BYTE#4 THEN
				X.ERROR_ID := ID;
			ELSE
				index := index + 2;
				BYTE_TO_BITS(IN:=X.R_BUF.BUFFER[index]);
				OUT1 := BYTE_TO_BITS.B0;
				OUT2 := BYTE_TO_BITS.B1;
				OUT3 := BYTE_TO_BITS.B2;
				OUT4 := BYTE_TO_BITS.B3;
				OUT5 := BYTE_TO_BITS.B4;
				OUT6 := BYTE_TO_BITS.B5;
				OUT7 := BYTE_TO_BITS.B6;
				OUT8 := BYTE_TO_BITS.B7;
				index := index + 1;
			END_IF;
		END_IF;
		X.index := index;
	END_IF;
END_IF;

(* revision history
ks	15.may. 2011	rev 1.0
	original version

*)

END_FUNCTION_BLOCK

// ---- oscat_basic/POUs/Logic/gate logic/BYTE_TO_BITS.TcPOU
FUNCTION_BLOCK BYTE_TO_BITS
VAR_INPUT
	IN: BYTE;
END_VAR
VAR_OUTPUT
	B0: BOOL;
	B1: BOOL;
	B2: BOOL;
	B3: BOOL;
	B4: BOOL;
	B5: BOOL;
	B6: BOOL;
	B7: BOOL;
END_VAR


(*
version 1.1	16. mar. 2008
programmer 	hugo
tested by		tobias

this Function Block extracts the 8 Bits from a byte


*)

B0 := IN.0;
B1 := IN.1;
B2 := IN.2;
B3 := IN.3;
B4 := IN.4;
B5 := IN.5;
B6 := IN.6;
B7 := IN.7;

(* revision history
hm		4. aug 2006	rev 1.0
	original version

hm		16. mar 2008	rev 1.1
	renamed from byte_to_bit to byte_to_bits for compatibility reasons

*)

END_FUNCTION_BLOCK

// ---- oscat_basic/POUs/Logic/gate logic/BYTE_OF_BIT.TcPOU
FUNCTION BYTE_OF_BIT : BYTE
VAR_INPUT
	B0:BOOL;
	B1:BOOL;
	B2:BOOL;
	B3:BOOL;
	B4:BOOL;
	B5:BOOL;
	B6:BOOL;
	B7:BOOL;
END_VAR


(*
version 1.1	 18. feb 2006
programmer 	hugo
tested by		tobias

this function creates a byte from 8 individual bits

*)

Byte_of_bit := SHL(SHL(SHL(SHL(SHL(SHL(SHL(BOOL_TO_BYTE(B7),1) OR BOOL_TO_BYTE(B6),1) OR BOOL_TO_BYTE(B5),1) OR BOOL_TO_BYTE(B4),1)
	OR BOOL_TO_BYTE(B3),1) OR BOOL_TO_BYTE(B2),1) OR BOOL_TO_BYTE(B1),1) OR BOOL_TO_BYTE(B0);


(* revision history

hm	4. aug 2006		rev 1.0
	original version

hm	18. feb. 2008	rev 1.1
	improved performance

*)

END_FUNCTION

// ---- beckhoff_network/POUs/NET_VAR/NET_VAR_STRING.TcPOU
FUNCTION_BLOCK NET_VAR_STRING
VAR_IN_OUT
	IN : STRING(STRING_LENGTH);
	OUT : STRING(STRING_LENGTH);
	X : NET_VAR_DATA;
END_VAR
VAR_OUTPUT
	ID : BYTE;
END_VAR
VAR
	init : BOOL;
	len_str : INT;
	index : INT;
	index2 : INT;
END_VAR

(*
version 1.0		15. may. 2011
programmer		ks
tested by			ks

NET_VAR_STRING überträgt bidirektional einen STRING vom Master zum Client
*)

IF NOT init THEN
	init := TRUE;
	X.ID_MAX := X.ID_MAX + USINT#1;
	ID := USINT_TO_BYTE(X.ID_MAX);
END_IF;

IF X.STATE > BYTE#0 AND X.ERROR_ID = BYTE#0 THEN
	index := X.index; (* PCWORX Workaround *)
	IF X.STATE = BYTE#1 THEN (* Daten schreiben *)
		len_str := LEN(IN);
		IF INT_TO_UINT(index + 3 + len_str) > X.BUF_SIZE THEN
			X.ERROR_ID := ID;
		ELSE
			X.S_BUF.BUFFER[index] := ID; (* ID *)
			index := index + 1;
			X.S_BUF.BUFFER[index] := BYTE#6; (* TYPE REAL *)
			index := index + 1;
			X.S_BUF.BUFFER[index] := INT_TO_BYTE(len_str); (* Anzahl der Bytes *)
			index := index + 1;
			_STRING_TO_BUFFER(STR:=IN,POS:=index,PT:=ADR(X.S_BUF.BUFFER),SIZE:=X.BUF_SIZE);
			index := index + len_str;
		END_IF;
	ELSIF X.STATE = BYTE#2 THEN (* Daten lesen *)
		index2 := index + 1; (* PCWORX Workaround *)
		IF X.R_BUF.BUFFER[index] <> ID OR X.R_BUF.BUFFER[index2] <> BYTE#6 THEN
			X.ERROR_ID := ID;
		ELSE
			index := index + 2;
			len_str := BYTE_TO_INT(X.R_BUF.BUFFER[index]);
			index2 := index + 1;
			index := index2 + len_str;
			IF len_STR > 0 THEN
				OUT := BUFFER_TO_STRING(PT:=ADR(X.R_BUF.BUFFER),SIZE:=X.BUF_SIZE,START:=INT_TO_UINT(index2),STOP:=INT_TO_UINT(index - 1));
			ELSE
				OUT := '';
			END_IF;
		END_IF;
	END_IF;
	X.index := index;
END_IF;

(* revision history
ks	15.may. 2011	rev 1.0
	original version

*)

END_FUNCTION_BLOCK

// ---- beckhoff_network/POUs/NET_VAR/NET_VAR_BUFFER.TcPOU
FUNCTION_BLOCK NET_VAR_BUFFER
VAR_IN_OUT
	BUF_IN : ARRAY[1..64] OF BYTE;
	BUF_OUT : ARRAY[1..64] OF BYTE;
	X : NET_VAR_DATA;
END_VAR
VAR_OUTPUT
	ID : BYTE;
END_VAR
VAR
	size : INT;
	init : BOOL;
	index : INT;
	index2 : INT;
END_VAR

(*
version 1.0		15. may. 2011
programmer		ks
tested by			ks

NET_VAR_BUFFER überträgt bidirektional 64 Bytes vom Master zum Client
*)

IF NOT init THEN
	init := TRUE;
	X.ID_MAX := X.ID_MAX + USINT#1;
	ID := USINT_TO_BYTE(X.ID_MAX);
END_IF;

IF X.STATE > BYTE#0 AND X.ERROR_ID = BYTE#0 THEN
	index := X.index; (* PCWORX Workaround *)
	IF X.STATE = BYTE#1 THEN (* Daten schreiben *)
		size := SIZEOF(BUF_IN);
		IF INT_TO_UINT(index + 3 + size) > X.BUF_SIZE THEN
			X.ERROR_ID := ID;
		ELSE
			X.S_BUF.BUFFER[index] := ID; (* ID *)
			index := index + 1;
			X.S_BUF.BUFFER[index] := BYTE#20; (* TYPE BUFFER *)
			index := index + 1;
			X.S_BUF.BUFFER[index] := INT_TO_BYTE(size); (* Anzahl der Bytes *)
				index := index + 1;
			FOR index2 := 1 TO size DO
				X.S_BUF.BUFFER[index] := BUF_IN[index2];
				index := index + 1;
			END_FOR;
		END_IF;
	ELSIF X.STATE = BYTE#2 THEN (* Daten lesen *)
		index2 := index + 1; (* PCWORX Workaround *)
		IF X.R_BUF.BUFFER[index] <> ID OR X.R_BUF.BUFFER[index2] <> BYTE#20 THEN
			X.ERROR_ID := ID;
		ELSE
			index := index + 2;
			size := BYTE_TO_INT(X.R_BUF.BUFFER[index]);
			index := index + 1;
			FOR index2 := 1 TO size DO
				BUF_OUT[index2] := X.R_BUF.BUFFER[index];
				index := index + 1;
			END_FOR;
		END_IF;
	END_IF;
	X.index := index;
END_IF;

(* revision history
ks	15.may. 2011	rev 1.0
	original version

*)

END_FUNCTION_BLOCK

// ---- beckhoff_network/POUs/NET_VAR/NET_VAR_DWORD8.TcPOU
FUNCTION_BLOCK NET_VAR_DWORD8
VAR_IN_OUT
	X : NET_VAR_DATA;
END_VAR
VAR_INPUT
	IN1 : DWORD;
	IN2 : DWORD;
	IN3 : DWORD;
	IN4 : DWORD;
	IN5 : DWORD;
	IN6 : DWORD;
	IN7 : DWORD;
	IN8 : DWORD;
END_VAR
VAR_OUTPUT
	OUT1 : DWORD;
	OUT2 : DWORD;
	OUT3 : DWORD;
	OUT4 : DWORD;
	OUT5 : DWORD;
	OUT6 : DWORD;
	OUT7 : DWORD;
	OUT8 : DWORD;
	ID : BYTE;
END_VAR
VAR
	init : BOOL;
	i : INT;
	i2 : INT;
	index : INT;
	index2 : INT;
	ra : ARRAY[1..8] OF DWORD;
END_VAR

(*
version 1.0		15. may. 2011
programmer		ks
tested by			ks

NET_VAR_DWORD8 überträgt bidirektional acht DWORD vom Master zum Client
*)

IF NOT init THEN
	init := TRUE;
	X.ID_MAX := X.ID_MAX + USINT#1;
	ID := USINT_TO_BYTE(X.ID_MAX);
END_IF;

IF X.STATE > BYTE#0 AND X.ERROR_ID = BYTE#0 THEN
	index := X.index; (* PCWORX Workaround *)
	IF INT_TO_UINT(index + 34) > X.BUF_SIZE THEN  (* ID (1) + TYPE (1) + 8 x DWORD (4) *)
		X.ERROR_ID := ID;
	ELSE
		IF X.STATE = BYTE#1 THEN (* Daten schreiben *)
			ra[1] := IN1;
			ra[2] := IN2;
			ra[3] := IN3;
			ra[4] := IN4;
			ra[5] := IN5;
			ra[6] := IN6;
			ra[7] := IN7;
			ra[8] := IN8;
			X.S_BUF.BUFFER[index] := ID; (* ID *)
			index := index + 1;
			X.S_BUF.BUFFER[index] := BYTE#13; (* TYPE DWORD8 *)
			index := index + 1;
			FOR i2 := 1 TO 8 DO;
				FOR i := 1 TO 4 DO;
					X.S_BUF.BUFFER[index] := DWORD_TO_BYTE(ra[i2]);
					ra[i2] := ROR(ra[i2],8);
					index := index + 1;
				END_FOR;
			END_FOR;

		ELSIF X.STATE = BYTE#2 THEN (* Daten lesen *)
			index2 := index + 1; (* PCWORX Workaround *)
			IF X.R_BUF.BUFFER[index] <> ID OR X.R_BUF.BUFFER[index2] <> BYTE#13 THEN (* TYPE DWORD8 *)
				X.ERROR_ID := ID;
			ELSE
				index := index + 2;
				FOR i2 := 1 TO 8 DO;
					ra[i2] := DWORD#0;
					FOR i := 1 TO 4 DO;
						ra[i2] := ra[i2] OR BYTE_TO_DWORD(X.R_BUF.BUFFER[index]);
						ra[i2] := ROR(ra[i2],8);
						index := index + 1;
					END_FOR;
				END_FOR;
				OUT1 := ra[1];
				OUT2 := ra[2];
				OUT3 := ra[3];
				OUT4 := ra[4];
				OUT5 := ra[5];
				OUT6 := ra[6];
				OUT7 := ra[7];
				OUT8 := ra[8];
			END_IF;
		END_IF;
		X.index := index;
	END_IF;
END_IF;

(* revision history
ks	15.may. 2011	rev 1.0
	original version

*)

END_FUNCTION_BLOCK

// ---- beckhoff_network/POUs/NET_VAR/NET_VAR_X8.TcPOU
FUNCTION_BLOCK NET_VAR_X8
VAR_IN_OUT
	X : NET_VAR_DATA;
END_VAR
VAR_INPUT
	IN_REAL1 : REAL;
	IN_REAL2 : REAL;
	IN_DINT1 : DINT;
	IN_DINT2 : DINT;
	IN_UDINT1 : UDINT;
	IN_UDINT2 : UDINT;
	IN_DWORD1 : DWORD;
	IN_DWORD2 : DWORD;
END_VAR
VAR_OUTPUT
	OUT_REAL1 : REAL;
	OUT_REAL2: REAL;
	OUT_DINT1 : DINT;
	OUT_DINT2 : DINT;
	OUT_UDINT1 : UDINT;
	OUT_UDINT2 : UDINT;
	OUT_DWORD1 : DWORD;
	OUT_DWORD2 : DWORD;
	ID : BYTE;
END_VAR
VAR
	init : BOOL;
	i : INT;
	i2 : INT;
	index : INT;
	index2 : INT;
	ra : ARRAY[1..8] OF DWORD;
END_VAR

(*
version 1.0		15. may. 2011
programmer		ks
tested by			ks

NET_VAR_X8 überträgt bidirektional 2x REAL,2x DINT,2x UDINT,2x DWORD vom Master zum Client
*)

IF NOT init THEN
	init := TRUE;
	X.ID_MAX := X.ID_MAX + USINT#1;
	ID := USINT_TO_BYTE(X.ID_MAX);
END_IF;

IF X.STATE > BYTE#0 AND X.ERROR_ID = BYTE#0 THEN
	index := X.index; (* PCWORX Workaround *)
	IF INT_TO_UINT(index + 34) > X.BUF_SIZE THEN  (* ID (1) + TYPE (1) + 8 x DWORD (4) *)
		X.ERROR_ID := ID;
	ELSE
		IF X.STATE = BYTE#1 THEN (* Daten schreiben *)
			ra[1] := REAL_TO_DW(X:=IN_REAL1);
			ra[2] := REAL_TO_DW(X:=IN_REAL2);
			ra[3] := DINT_TO_DWORD(IN_DINT1);
			ra[4] := DINT_TO_DWORD(IN_DINT2);
			ra[5] := UDINT_TO_DWORD(IN_UDINT1);
			ra[6] := UDINT_TO_DWORD(IN_UDINT2);
			ra[7] := IN_DWORD1;
			ra[8] := IN_DWORD2;
			X.S_BUF.BUFFER[index] := ID; (* ID *)
			index := index + 1;
			X.S_BUF.BUFFER[index] := BYTE#21; (* TYPE X8 *)
			index := index + 1;
			FOR i2 := 1 TO 8 DO;
				FOR i := 1 TO 4 DO;
					X.S_BUF.BUFFER[index] := DWORD_TO_BYTE(ra[i2]);
					ra[i2] := ROR(ra[i2],8);
					index := index + 1;
				END_FOR;
			END_FOR;

		ELSIF X.STATE = BYTE#2 THEN (* Daten lesen *)
			index2 := index + 1; (* PCWORX Workaround *)
			IF X.R_BUF.BUFFER[index] <> ID OR X.R_BUF.BUFFER[index2] <> BYTE#21 THEN (* TYPE X8 *)
				X.ERROR_ID := ID;
			ELSE
				index := index + 2;
				FOR i2 := 1 TO 8 DO;
					ra[i2] := DWORD#0;
					FOR i := 1 TO 4 DO;
						ra[i2] := ra[i2] OR BYTE_TO_DWORD(X.R_BUF.BUFFER[index]);
						ra[i2] := ROR(ra[i2],8);
						index := index + 1;
					END_FOR;
				END_FOR;
				OUT_REAL1 := DW_TO_REAL(X:=ra[1]);
				OUT_REAL2 := DW_TO_REAL(X:=ra[2]);
				OUT_DINT1 := DWORD_TO_DINT(ra[3]);
				OUT_DINT2 := DWORD_TO_DINT(ra[4]);
				OUT_UDINT1 := DWORD_TO_UDINT(ra[5]);
				OUT_UDINT2 := DWORD_TO_UDINT(ra[6]);
				OUT_DWORD1 := ra[7];
				OUT_DWORD2 := ra[8];
			END_IF;
		END_IF;
		X.index := index;
	END_IF;
END_IF;

(* revision history
ks	15.may. 2011	rev 1.0
	original version

*)

END_FUNCTION_BLOCK

// ---- beckhoff_network/POUs/DEMO/SHA1_MD5_DEMO.TcPOU
PROGRAM SHA1_MD5_DEMO
VAR
	text: STRING(STRING_LENGTH) := '<4036.1076324381@guildenstern.zeitform.de>';
	MD5_STR : MD5_STR;
	SHA1_STR : SHA1_STR;
	md5_hash : ARRAY [0..15] OF BYTE;
	sha1_hash : ARRAY [0..19] OF BYTE;
	start1 : BOOL := TRUE;
	start2 : BOOL := TRUE;
	done1 : BOOL;
	done2 : BOOL;
	md5_strh : STRING(32);
	sha1_strh : STRING(40);
END_VAR

MD5_STR(RUN := start1, STR := text, MD5 := md5_hash);
done1 := MD5_STR.DONE;
md5_strh := MD5_TO_STRH(MD5 := md5_hash);
SHA1_STR(RUN := start2, STR := text, SHA1 := sha1_hash);
done2 := SHA1_STR.DONE;
sha1_strh := SHA1_TO_STRH(SHA1 := sha1_hash);

END_PROGRAM

// ---- beckhoff_network/POUs/DEMO/SMTP_CLIENT_DEMO.TcPOU
PROGRAM SMTP_CLIENT_DEMO
VAR
(*
	smtp_server: STRING := 'oscat_test%freenet.de:oscat123456@mx.freenet.de';
	smtp_mailfrom: STRING := 'oscat_test@freenet.de';
*)

	SMTP_CLIENT: SMTP_CLIENT;
	smtp_activate: BOOL;
	smtp_timeout: TIME := T#30s;
	smtp_error_t: BYTE;
	smtp_error_c: DWORD;
	smtp_busy: BOOL;
	smtp_done: BOOL;
	smtp_dti: DT;
	smtp_dti_offset: INT := 60;
	smtp_files: STRING(STRING_LENGTH) := '';
	smtp_server: STRING := '110876022:oscat123456@mail.gmx.net';
	smtp_mailfrom: STRING := 'oscat@gmx.net;Station_01';
	smtp_mailto: STRING(STRING_LENGTH) := 'oscat@gmx.net';
	smtp_subject: STRING := 'Das ist der Betreff';
	smtp_body: STRING(STRING_LENGTH) := 'Das ist der Email-Text';
END_VAR
VAR // added by the converter: edge detectors and wires of the graphical bodies
    _w1 : ANY;
END_VAR

_w1 := DWORD_OF_BYTE(8, 8, 8, 8);
SMTP_CLIENT(
    ACTIVATE := smtp_activate,
    TIMEOUT := smtp_timeout,
    DTI := smtp_dti,
    DTI_OFFSET := smtp_dti_offset,
    DNS_IP4 := _w1,
    SERVER := smtp_server,
    MAILFROM := smtp_mailfrom,
    MAILTO := smtp_mailto,
    SUBJECT := smtp_subject,
    BODY := smtp_body,
    FILES := smtp_files);
smtp_done := SMTP_CLIENT.DONE;
smtp_busy := SMTP_CLIENT.BUSY;
smtp_error_c := SMTP_CLIENT.ERROR_C;
smtp_error_t := SMTP_CLIENT.ERROR_T;

END_PROGRAM

// ---- beckhoff_network/POUs/NETWORK/SMTP_CLIENT.TcPOU
FUNCTION_BLOCK SMTP_CLIENT
VAR_INPUT
	ACTIVATE : BOOL;
	TIMEOUT : TIME;
	DTI : DT;
	DTI_OFFSET : INT;
	DNS_IP4 : DWORD;
END_VAR
VAR_OUTPUT
	DONE : BOOL;
	BUSY : BOOL;
	ERROR_C : DWORD;
	ERROR_T : BYTE;
END_VAR
VAR_IN_OUT
	SERVER : STRING;
	MAILFROM : STRING;
	MAILTO : STRING(STRING_LENGTH);
	SUBJECT : STRING;
	BODY : STRING(STRING_LENGTH);
	FILES : STRING(STRING_LENGTH);
END_VAR
VAR
	IP_C : IP_C; (* IP_Control Verwaltungsstruktur *)
	S_BUF : NETWORK_BUFFER;
	R_BUF : NETWORK_BUFFER;
	F_BUF : NETWORK_BUFFER;
	URL_DATA : url;
	DNS_CLIENT : DNS_CLIENT;
	IPC : IP_CONTROL;
	FS : FILE_SERVER;
	FSD : FILE_SERVER_DATA;
	BASE64_ENCODE_STR : BASE64_ENCODE_STR;
	BASE64_ENCODE_STREAM : BASE64_ENCODE_STREAM;
	fpd : FILE_PATH_DATA;
	MD5_CRAM_AUTH : MD5_CRAM_AUTH;
	MD5_RUN : BOOL;
	activate_last : BOOL;
	step : INT;
	snd_step : INT;
	str1 : STRING(STRING_LENGTH);
	str2 : STRING(STRING_LENGTH);
	str3 : STRING;
	snd_text :	STRING(STRING_LENGTH);
	snd_lf_cnt : INT;
	rcv_text :	STRING(STRING_LENGTH);
	rcv_s : STRING(3);
	rcv_state : INT;
	auth_names : STRING := ' PLAIN; LOGIN; CRAM-MD5';
	auth_state : BYTE;
	TON_WAIT : TON;
	last_step : INT;
	next_step : INT;
	timeout2 : TIME;
	timeout3 : TIME;
	last_block : BOOL;
	file_delete : BOOL;
	esmtp : BOOL;
	cnt1 : INT;
	cnt2 : INT;
	cnt3 : INT;
	cnt4 : INT;
	idx1 : INT;
	idx2 : INT;
	idx3 : INT;
	snd_idx : INT;
	snd_enable : BOOL;
	i1 : INT;
	b64_done : BOOL;
	b64_start : BOOL;
	b64_max : UINT := 2880; (* short = 960 / long = 2880 *)
	b64_buf1 : ARRAY [0..47] OF BYTE;
	b64_buf2 : ARRAY [0..63] OF BYTE;
	b64_size1 : INT;
	b64_size2 : INT;
	b64_lf : BOOL;
	b64_str1	: STRING(144);
	b64_str2	: STRING(192);
	md5_user : STRING(64);
	md5_password : STRING(64);
	md5_b64_ts : STRING(64);
	md5_auth_key : STRING(192);
	ip_c_red_disable : BOOL; (* IP_CONTROL - Remote Disconnect Error unterdrücken *)

	(*LOG_MSG : LOG_MSG;
	_debug_enable : BOOL := TRUE;*)
END_VAR

(*
version 1.3		30. may 2011
programmer		ks
tested by			ks

SMTP_CLIENT versendet Email an verschiedene Emailadressen mit optionalen Dateianhängen.



mögliche Rückgabecodes:

Grad der Schwere
 
Die erste Stelle des Rückgabecodes gibt den Grad der Schwere an:
1yz Vorläufige positive Antwort
2yz Antwort über positiven Abschluss 
3yz Positive Zwischenantwort 
4yz Antwort über vorübergehenden negativen Abschluss 
5yz Permanente negative Antwort 
 
Die zweite Stelle gibt die Kategorie der Antwort an: 
x0z Syntaxfehler 
x1z Information 
x2z Verbindung 
x3z Nicht festgelegt 
x4z Nicht festgelegt 
x5z Mail-System 
 
Die dritte Stelle dient zur genaueren Bestimmung der Kategorie. 

